// Mitsubishi GX Works2 project: 1 A22-0150 PLC_230728   PLC: Q03UDV

PROGRAM 001  // 現在値ｶｳﾝﾄ
      P100
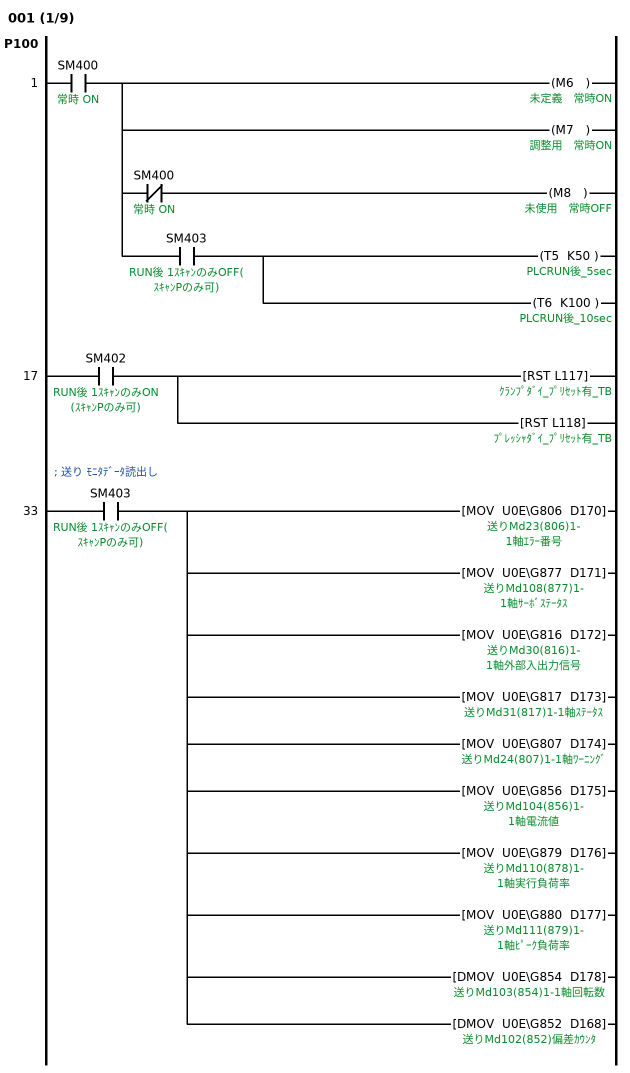
1     LD      SM400  ; 常時 ON
      OUT     M6  ; 未定義　常時ON
      OUT     M7  ; 調整用　常時ON
      MPS
      ANI     SM400  ; 常時 ON
      OUT     M8  ; 未使用　常時OFF
      MPP
      AND     SM403  ; RUN後 1ｽｷｬﾝのみOFF(ｽｷｬﾝPのみ可)
      OUT     T5 K50  ; PLCRUN後_5sec
      OUT     T6 K100  ; PLCRUN後_10sec
17    LD      SM402  ; RUN後 1ｽｷｬﾝのみON (ｽｷｬﾝPのみ可)
      RST     L117  ; ｸﾗﾝﾌﾟﾀﾞｲ_ﾌﾟﾘｾｯﾄ有_TB
      RST     L118  ; ﾌﾟﾚｯｼｬﾀﾞｲ_ﾌﾟﾘｾｯﾄ有_TB
; 
; 送り ﾓﾆﾀﾃﾞｰﾀ読出し
33    LD      SM403  ; RUN後 1ｽｷｬﾝのみOFF(ｽｷｬﾝPのみ可)
      MOV     U0E\G806 D170  ; 送りMd23(806)1-1軸ｴﾗｰ番号
      MOV     U0E\G877 D171  ; 送りMd108(877)1-1軸ｻｰﾎﾞｽﾃｰﾀｽ
      MOV     U0E\G816 D172  ; 送りMd30(816)1-1軸外部入出力信号
      MOV     U0E\G817 D173  ; 送りMd31(817)1-1軸ｽﾃｰﾀｽ
      MOV     U0E\G807 D174  ; 送りMd24(807)1-1軸ﾜｰﾆﾝｸﾞ
      MOV     U0E\G856 D175  ; 送りMd104(856)1-1軸電流値
      MOV     U0E\G879 D176  ; 送りMd110(878)1-1軸実行負荷率
      MOV     U0E\G880 D177  ; 送りMd111(879)1-1軸ﾋﾟｰｸ負荷率
      DMOV    U0E\G854 D178  ; 送りMd103(854)1-1軸回転数
      DMOV    U0E\G852 D168  ; 送りMd102(852)偏差ｶｳﾝﾀ
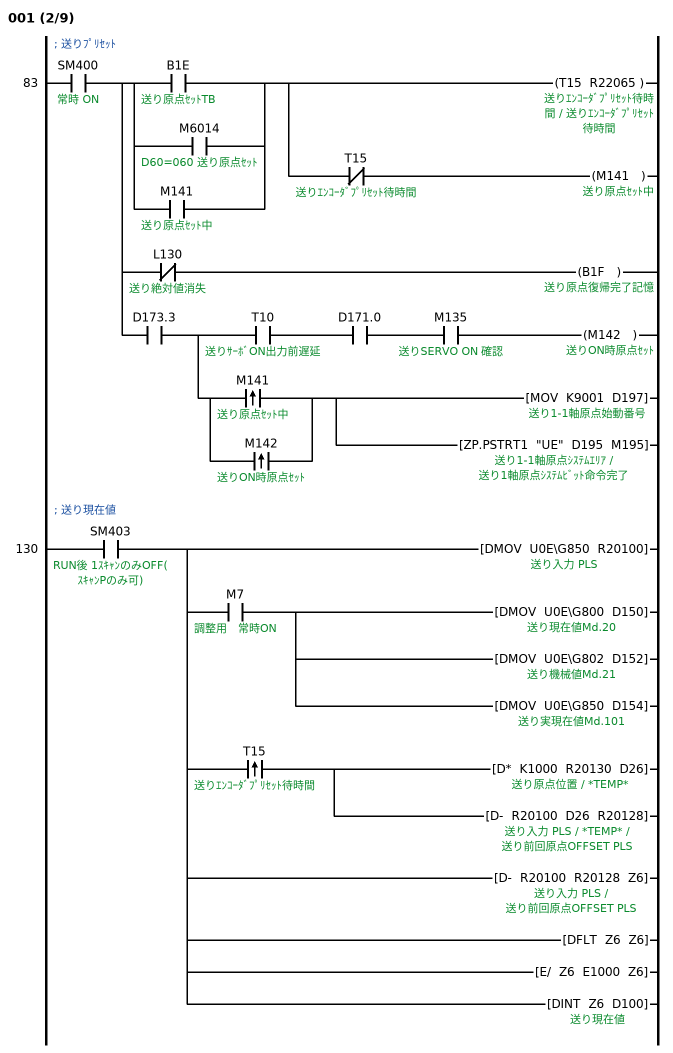
; 
; 送りﾌﾟﾘｾｯﾄ
83    LD      SM400  ; 常時 ON
      MPS
      LD      B1E  ; 送り原点ｾｯﾄTB
      OR      M6014  ; D60=060 送り原点ｾｯﾄ
      OR      M141  ; 送り原点ｾｯﾄ中
      ANB
      OUT     T15 R22065  ; 送りｴﾝｺｰﾀﾞﾌﾟﾘｾｯﾄ待時間 / 送りｴﾝｺｰﾀﾞﾌﾟﾘｾｯﾄ待時間
      ANI     T15  ; 送りｴﾝｺｰﾀﾞﾌﾟﾘｾｯﾄ待時間
      OUT     M141  ; 送り原点ｾｯﾄ中
      MRD
      ANI     L130  ; 送り絶対値消失
      OUT     B1F  ; 送り原点復帰完了記憶
      MPP
      AND     D173.3
      MPS
      AND     T10  ; 送りｻｰﾎﾞON出力前遅延
      AND     D171.0
      AND     M135  ; 送りSERVO ON 確認
      OUT     M142  ; 送りON時原点ｾｯﾄ
      MPP
      LDP     M141  ; 送り原点ｾｯﾄ中
      ORP     M142  ; 送りON時原点ｾｯﾄ
      ANB
      MOV     K9001 D197  ; 送り1-1軸原点始動番号
      ZP.PSTRT1 "UE" D195 M195  ; 送り1-1軸原点ｼｽﾃﾑｴﾘｱ / 送り1軸原点ｼｽﾃﾑﾋﾞｯﾄ命令完了
; 送り現在値
130   LD      SM403  ; RUN後 1ｽｷｬﾝのみOFF(ｽｷｬﾝPのみ可)
      DMOV    U0E\G850 R20100  ; 送り入力 PLS
      MPS
      AND     M7  ; 調整用　常時ON
      DMOV    U0E\G800 D150  ; 送り現在値Md.20
      DMOV    U0E\G802 D152  ; 送り機械値Md.21
      DMOV    U0E\G850 D154  ; 送り実現在値Md.101
      MRD
      ANDP    T15  ; 送りｴﾝｺｰﾀﾞﾌﾟﾘｾｯﾄ待時間
      D*      K1000 R20130 D26  ; 送り原点位置 / *TEMP*
      D-      R20100 D26 R20128  ; 送り前回原点OFFSET PLS
      MPP
      D-      R20100 R20128 Z6
      DFLT    Z6 Z6
      E/      Z6 E1000 Z6
      DINT    Z6 D100  ; 送り現在値
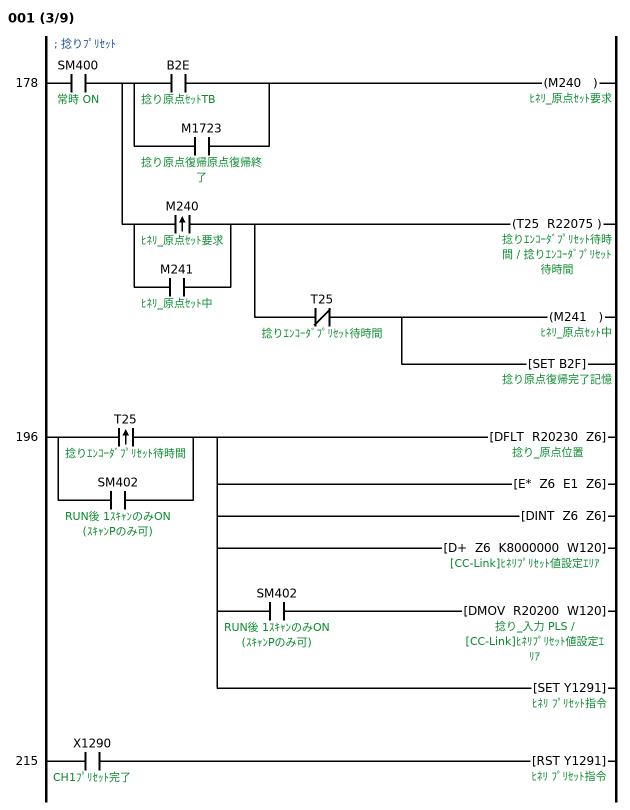
; 
; 捻りﾌﾟﾘｾｯﾄ
178   LD      SM400  ; 常時 ON
      MPS
      LD      B2E  ; 捻り原点ｾｯﾄTB
      OR      M1723  ; 捻り原点復帰原点復帰終了
      ANB
      OUT     M240  ; ﾋﾈﾘ_原点ｾｯﾄ要求
      MPP
      LDP     M240  ; ﾋﾈﾘ_原点ｾｯﾄ要求
      OR      M241  ; ﾋﾈﾘ_原点ｾｯﾄ中
      ANB
      OUT     T25 R22075  ; 捻りｴﾝｺｰﾀﾞﾌﾟﾘｾｯﾄ待時間 / 捻りｴﾝｺｰﾀﾞﾌﾟﾘｾｯﾄ待時間
      ANI     T25  ; 捻りｴﾝｺｰﾀﾞﾌﾟﾘｾｯﾄ待時間
      OUT     M241  ; ﾋﾈﾘ_原点ｾｯﾄ中
      SET     B2F  ; 捻り原点復帰完了記憶
196   LDP     T25  ; 捻りｴﾝｺｰﾀﾞﾌﾟﾘｾｯﾄ待時間
      OR      SM402  ; RUN後 1ｽｷｬﾝのみON (ｽｷｬﾝPのみ可)
      DFLT    R20230 Z6  ; 捻り_原点位置
      E*      Z6 E1 Z6
      DINT    Z6 Z6
      D+      Z6 K8000000 W120  ; [CC-Link]ﾋﾈﾘﾌﾟﾘｾｯﾄ値設定ｴﾘｱ
      MPS
      AND     SM402  ; RUN後 1ｽｷｬﾝのみON (ｽｷｬﾝPのみ可)
      DMOV    R20200 W120  ; 捻り_入力 PLS
      MPP
      SET     Y1291  ; ﾋﾈﾘ ﾌﾟﾘｾｯﾄ指令
215   LD      X1290  ; CH1ﾌﾟﾘｾｯﾄ完了
      RST     Y1291  ; ﾋﾈﾘ ﾌﾟﾘｾｯﾄ指令
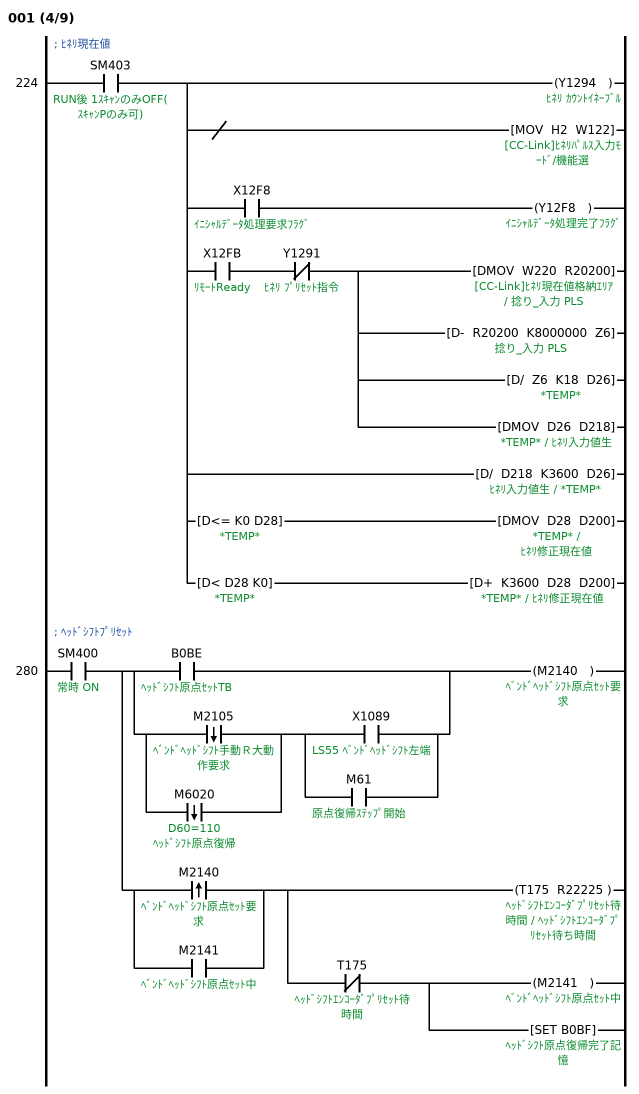
; ﾋﾈﾘ現在値
224   LD      SM403  ; RUN後 1ｽｷｬﾝのみOFF(ｽｷｬﾝPのみ可)
      OUT     Y1294  ; ﾋﾈﾘ ｶｳﾝﾄｲﾈｰﾌﾞﾙ
      MPS
      INV
      MOV     H2 W122  ; [CC-Link]ﾋﾈﾘﾊﾟﾙｽ入力ﾓｰﾄﾞ/機能選
      MRD
      AND     X12F8  ; ｲﾆｼｬﾙﾃﾞｰﾀ処理要求ﾌﾗｸﾞ
      OUT     Y12F8  ; ｲﾆｼｬﾙﾃﾞｰﾀ処理完了ﾌﾗｸﾞ
      MRD
      AND     X12FB  ; ﾘﾓｰﾄReady
      ANI     Y1291  ; ﾋﾈﾘ ﾌﾟﾘｾｯﾄ指令
      DMOV    W220 R20200  ; [CC-Link]ﾋﾈﾘ現在値格納ｴﾘｱ
      D-      R20200 K8000000 Z6
      D/      Z6 K18 D26
      DMOV    D26 D218  ; ﾋﾈﾘ入力値生
      MPP
      D/      D218 K3600 D26
      MPS
      ANDD<=  K0 D28  ; *TEMP*
      DMOV    D28 D200  ; ﾋﾈﾘ修正現在値
      MPP
      ANDD<   D28 K0  ; *TEMP*
      D+      K3600 D28 D200
; 
; ﾍｯﾄﾞｼﾌﾄﾌﾟﾘｾｯﾄ
280   LD      SM400  ; 常時 ON
      MPS
      LD      B0BE  ; ﾍｯﾄﾞｼﾌﾄ原点ｾｯﾄTB
      LDF     M2105  ; ﾍﾞﾝﾄﾞﾍｯﾄﾞｼﾌﾄ手動Ｒ大動作要求
      ORF     M6020  ; D60=110 ﾍｯﾄﾞｼﾌﾄ原点復帰
      LD      X1089  ; LS55 ﾍﾞﾝﾄﾞﾍｯﾄﾞｼﾌﾄ左端
      OR      M61  ; 原点復帰ｽﾃｯﾌﾟ開始
      ANB
      ORB
      ANB
      OUT     M2140  ; ﾍﾞﾝﾄﾞﾍｯﾄﾞｼﾌﾄ原点ｾｯﾄ要求
      MPP
      LDP     M2140  ; ﾍﾞﾝﾄﾞﾍｯﾄﾞｼﾌﾄ原点ｾｯﾄ要求
      OR      M2141  ; ﾍﾞﾝﾄﾞﾍｯﾄﾞｼﾌﾄ原点ｾｯﾄ中
      ANB
      OUT     T175 R22225  ; ﾍｯﾄﾞｼﾌﾄｴﾝｺｰﾀﾞﾌﾟﾘｾｯﾄ待時間 / ﾍｯﾄﾞｼﾌﾄｴﾝｺｰﾀﾞﾌﾟﾘｾｯﾄ待ち時間
      ANI     T175  ; ﾍｯﾄﾞｼﾌﾄｴﾝｺｰﾀﾞﾌﾟﾘｾｯﾄ待時間
      OUT     M2141  ; ﾍﾞﾝﾄﾞﾍｯﾄﾞｼﾌﾄ原点ｾｯﾄ中
      SET     B0BF  ; ﾍｯﾄﾞｼﾌﾄ原点復帰完了記憶
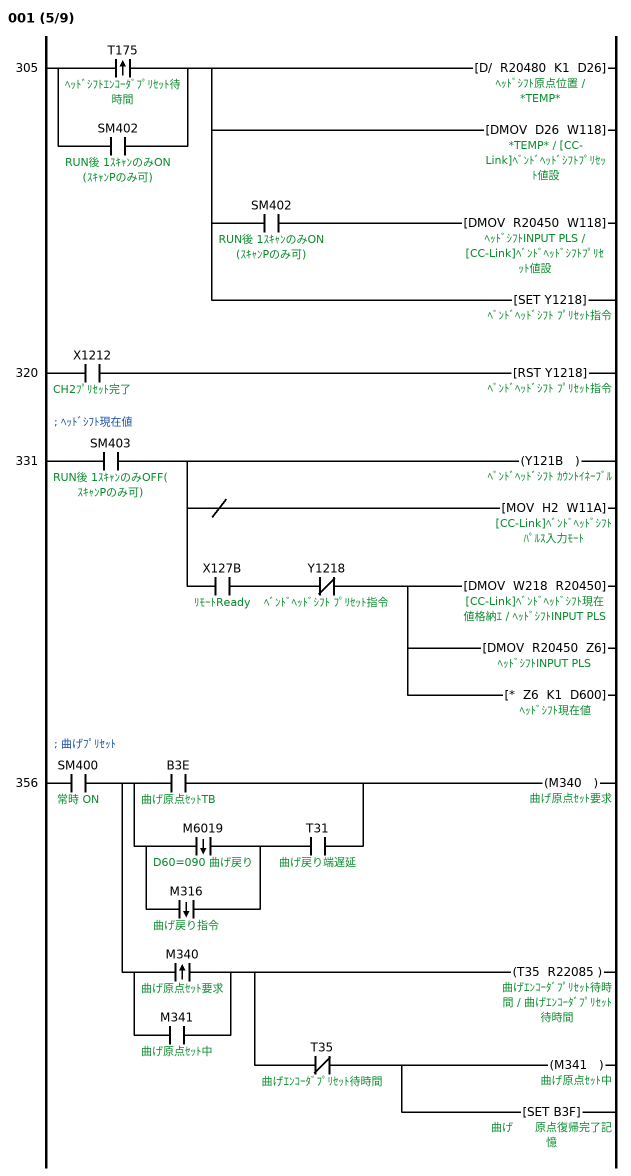
305   LDP     T175  ; ﾍｯﾄﾞｼﾌﾄｴﾝｺｰﾀﾞﾌﾟﾘｾｯﾄ待時間
      OR      SM402  ; RUN後 1ｽｷｬﾝのみON (ｽｷｬﾝPのみ可)
      D/      R20480 K1 D26  ; ﾍｯﾄﾞｼﾌﾄ原点位置
      DMOV    D26 W118  ; [CC-Link]ﾍﾞﾝﾄﾞﾍｯﾄﾞｼﾌﾄﾌﾟﾘｾｯﾄ値設
      MPS
      AND     SM402  ; RUN後 1ｽｷｬﾝのみON (ｽｷｬﾝPのみ可)
      DMOV    R20450 W118  ; ﾍｯﾄﾞｼﾌﾄINPUT PLS
      MPP
      SET     Y1218  ; ﾍﾞﾝﾄﾞﾍｯﾄﾞｼﾌﾄ ﾌﾟﾘｾｯﾄ指令
320   LD      X1212  ; CH2ﾌﾟﾘｾｯﾄ完了
      RST     Y1218  ; ﾍﾞﾝﾄﾞﾍｯﾄﾞｼﾌﾄ ﾌﾟﾘｾｯﾄ指令
; ﾍｯﾄﾞｼﾌﾄ現在値
331   LD      SM403  ; RUN後 1ｽｷｬﾝのみOFF(ｽｷｬﾝPのみ可)
      OUT     Y121B  ; ﾍﾞﾝﾄﾞﾍｯﾄﾞｼﾌﾄ ｶｳﾝﾄｲﾈｰﾌﾞﾙ
      MPS
      INV
      MOV     H2 W11A  ; [CC-Link]ﾍﾞﾝﾄﾞﾍｯﾄﾞｼﾌﾄﾊﾟﾙｽ入力ﾓｰﾄ
      MPP
      AND     X127B  ; ﾘﾓｰﾄReady
      ANI     Y1218  ; ﾍﾞﾝﾄﾞﾍｯﾄﾞｼﾌﾄ ﾌﾟﾘｾｯﾄ指令
      DMOV    W218 R20450  ; [CC-Link]ﾍﾞﾝﾄﾞﾍｯﾄﾞｼﾌﾄ現在値格納ｴ
      DMOV    R20450 Z6
      *       Z6 K1 D600  ; ﾍｯﾄﾞｼﾌﾄ現在値
; 
; 曲げﾌﾟﾘｾｯﾄ
356   LD      SM400  ; 常時 ON
      MPS
      LD      B3E  ; 曲げ原点ｾｯﾄTB
      LDF     M6019  ; D60=090 曲げ戻り
      ORF     M316  ; 曲げ戻り指令
      AND     T31  ; 曲げ戻り端遅延
      ORB
      ANB
      OUT     M340  ; 曲げ原点ｾｯﾄ要求
      MPP
      LDP     M340  ; 曲げ原点ｾｯﾄ要求
      OR      M341  ; 曲げ原点ｾｯﾄ中
      ANB
      OUT     T35 R22085  ; 曲げｴﾝｺｰﾀﾞﾌﾟﾘｾｯﾄ待時間 / 曲げｴﾝｺｰﾀﾞﾌﾟﾘｾｯﾄ待時間
      ANI     T35  ; 曲げｴﾝｺｰﾀﾞﾌﾟﾘｾｯﾄ待時間
      OUT     M341  ; 曲げ原点ｾｯﾄ中
      SET     B3F  ; 曲げ　　原点復帰完了記憶
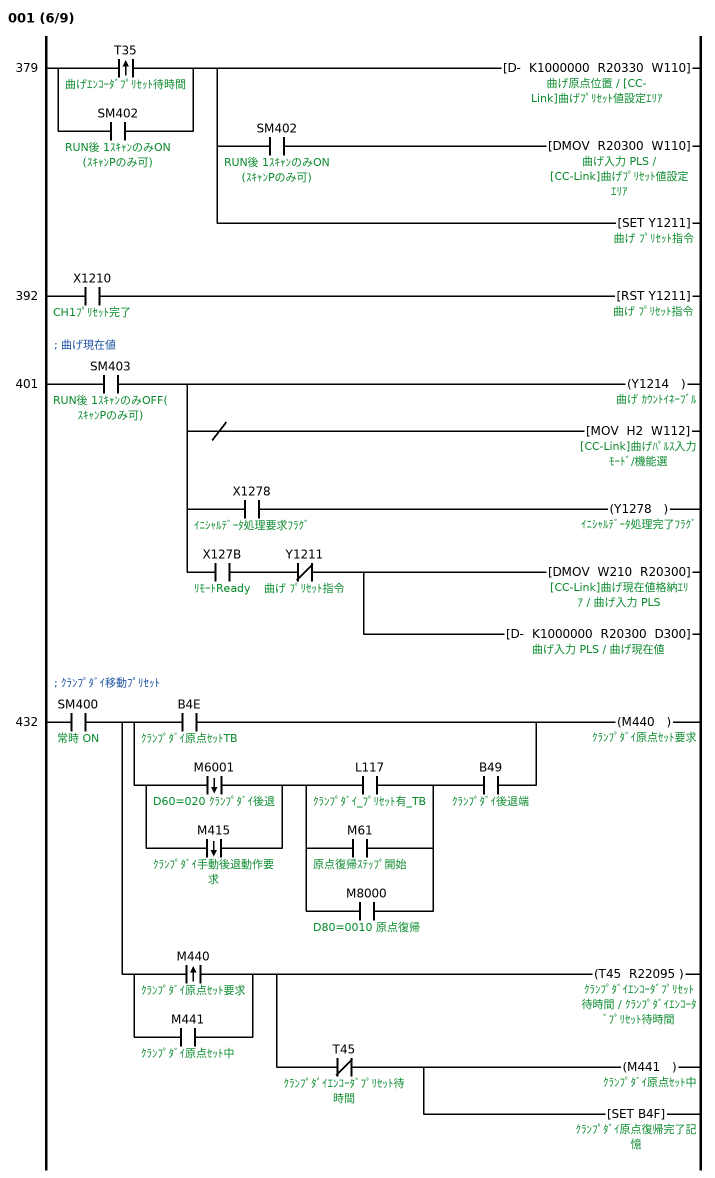
379   LDP     T35  ; 曲げｴﾝｺｰﾀﾞﾌﾟﾘｾｯﾄ待時間
      OR      SM402  ; RUN後 1ｽｷｬﾝのみON (ｽｷｬﾝPのみ可)
      D-      K1000000 R20330 W110  ; 曲げ原点位置 / [CC-Link]曲げﾌﾟﾘｾｯﾄ値設定ｴﾘｱ
      MPS
      AND     SM402  ; RUN後 1ｽｷｬﾝのみON (ｽｷｬﾝPのみ可)
      DMOV    R20300 W110  ; 曲げ入力 PLS
      MPP
      SET     Y1211  ; 曲げ ﾌﾟﾘｾｯﾄ指令
392   LD      X1210  ; CH1ﾌﾟﾘｾｯﾄ完了
      RST     Y1211  ; 曲げ ﾌﾟﾘｾｯﾄ指令
; 曲げ現在値
401   LD      SM403  ; RUN後 1ｽｷｬﾝのみOFF(ｽｷｬﾝPのみ可)
      OUT     Y1214  ; 曲げ ｶｳﾝﾄｲﾈｰﾌﾞﾙ
      MPS
      INV
      MOV     H2 W112  ; [CC-Link]曲げﾊﾟﾙｽ入力ﾓｰﾄﾞ/機能選
      MRD
      AND     X1278  ; ｲﾆｼｬﾙﾃﾞｰﾀ処理要求ﾌﾗｸﾞ
      OUT     Y1278  ; ｲﾆｼｬﾙﾃﾞｰﾀ処理完了ﾌﾗｸﾞ
      MPP
      AND     X127B  ; ﾘﾓｰﾄReady
      ANI     Y1211  ; 曲げ ﾌﾟﾘｾｯﾄ指令
      DMOV    W210 R20300  ; [CC-Link]曲げ現在値格納ｴﾘｱ
      D-      K1000000 R20300 D300  ; 曲げ現在値
; 
; ｸﾗﾝﾌﾟﾀﾞｲ移動ﾌﾟﾘｾｯﾄ
432   LD      SM400  ; 常時 ON
      MPS
      LD      B4E  ; ｸﾗﾝﾌﾟﾀﾞｲ原点ｾｯﾄTB
      LDF     M6001  ; D60=020 ｸﾗﾝﾌﾟﾀﾞｲ後退
      ORF     M415  ; ｸﾗﾝﾌﾟﾀﾞｲ手動後退動作要求
      LD      L117  ; ｸﾗﾝﾌﾟﾀﾞｲ_ﾌﾟﾘｾｯﾄ有_TB
      OR      M61  ; 原点復帰ｽﾃｯﾌﾟ開始
      OR      M8000  ; D80=0010 原点復帰
      ANB
      AND     B49  ; ｸﾗﾝﾌﾟﾀﾞｲ後退端
      ORB
      ANB
      OUT     M440  ; ｸﾗﾝﾌﾟﾀﾞｲ原点ｾｯﾄ要求
      MPP
      LDP     M440  ; ｸﾗﾝﾌﾟﾀﾞｲ原点ｾｯﾄ要求
      OR      M441  ; ｸﾗﾝﾌﾟﾀﾞｲ原点ｾｯﾄ中
      ANB
      OUT     T45 R22095  ; ｸﾗﾝﾌﾟﾀﾞｲｴﾝｺｰﾀﾞﾌﾟﾘｾｯﾄ待時間 / ｸﾗﾝﾌﾟﾀﾞｲｴﾝｺｰﾀﾞﾌﾟﾘｾｯﾄ待時間
      ANI     T45  ; ｸﾗﾝﾌﾟﾀﾞｲｴﾝｺｰﾀﾞﾌﾟﾘｾｯﾄ待時間
      OUT     M441  ; ｸﾗﾝﾌﾟﾀﾞｲ原点ｾｯﾄ中
      SET     B4F  ; ｸﾗﾝﾌﾟﾀﾞｲ原点復帰完了記憶
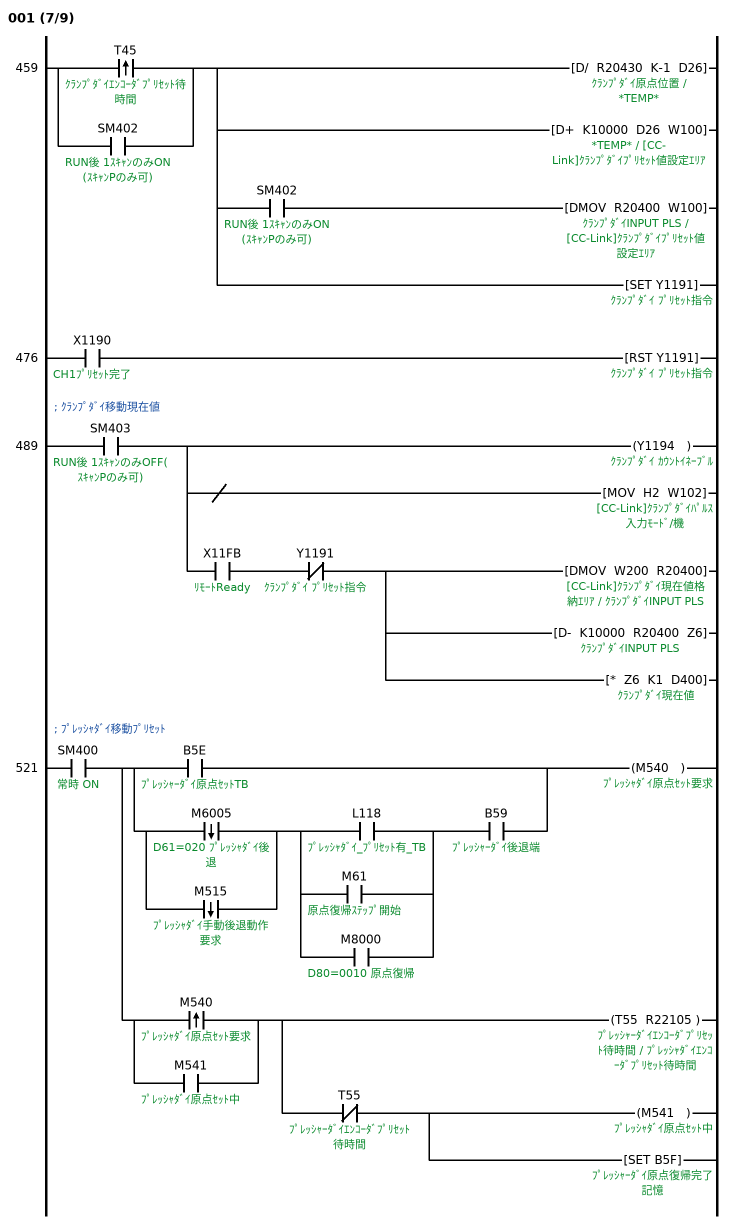
459   LDP     T45  ; ｸﾗﾝﾌﾟﾀﾞｲｴﾝｺｰﾀﾞﾌﾟﾘｾｯﾄ待時間
      OR      SM402  ; RUN後 1ｽｷｬﾝのみON (ｽｷｬﾝPのみ可)
      D/      R20430 K-1 D26  ; ｸﾗﾝﾌﾟﾀﾞｲ原点位置
      D+      K10000 D26 W100  ; [CC-Link]ｸﾗﾝﾌﾟﾀﾞｲﾌﾟﾘｾｯﾄ値設定ｴﾘｱ
      MPS
      AND     SM402  ; RUN後 1ｽｷｬﾝのみON (ｽｷｬﾝPのみ可)
      DMOV    R20400 W100  ; ｸﾗﾝﾌﾟﾀﾞｲINPUT PLS
      MPP
      SET     Y1191  ; ｸﾗﾝﾌﾟﾀﾞｲ ﾌﾟﾘｾｯﾄ指令
476   LD      X1190  ; CH1ﾌﾟﾘｾｯﾄ完了
      RST     Y1191  ; ｸﾗﾝﾌﾟﾀﾞｲ ﾌﾟﾘｾｯﾄ指令
; ｸﾗﾝﾌﾟﾀﾞｲ移動現在値
489   LD      SM403  ; RUN後 1ｽｷｬﾝのみOFF(ｽｷｬﾝPのみ可)
      OUT     Y1194  ; ｸﾗﾝﾌﾟﾀﾞｲ ｶｳﾝﾄｲﾈｰﾌﾞﾙ
      MPS
      INV
      MOV     H2 W102  ; [CC-Link]ｸﾗﾝﾌﾟﾀﾞｲﾊﾟﾙｽ入力ﾓｰﾄﾞ/機
      MPP
      AND     X11FB  ; ﾘﾓｰﾄReady
      ANI     Y1191  ; ｸﾗﾝﾌﾟﾀﾞｲ ﾌﾟﾘｾｯﾄ指令
      DMOV    W200 R20400  ; [CC-Link]ｸﾗﾝﾌﾟﾀﾞｲ現在値格納ｴﾘｱ
      D-      K10000 R20400 Z6
      *       Z6 K1 D400  ; ｸﾗﾝﾌﾟﾀﾞｲ現在値
; 
; ﾌﾟﾚｯｼｬﾀﾞｲ移動ﾌﾟﾘｾｯﾄ
521   LD      SM400  ; 常時 ON
      MPS
      LD      B5E  ; ﾌﾟﾚｯｼｬｰﾀﾞｲ原点ｾｯﾄTB
      LDF     M6005  ; D61=020 ﾌﾟﾚｯｼｬﾀﾞｲ後退
      ORF     M515  ; ﾌﾟﾚｯｼｬﾀﾞｲ手動後退動作要求
      LD      L118  ; ﾌﾟﾚｯｼｬﾀﾞｲ_ﾌﾟﾘｾｯﾄ有_TB
      OR      M61  ; 原点復帰ｽﾃｯﾌﾟ開始
      OR      M8000  ; D80=0010 原点復帰
      ANB
      AND     B59  ; ﾌﾟﾚｯｼｬｰﾀﾞｲ後退端
      ORB
      ANB
      OUT     M540  ; ﾌﾟﾚｯｼｬﾀﾞｲ原点ｾｯﾄ要求
      MPP
      LDP     M540  ; ﾌﾟﾚｯｼｬﾀﾞｲ原点ｾｯﾄ要求
      OR      M541  ; ﾌﾟﾚｯｼｬﾀﾞｲ原点ｾｯﾄ中
      ANB
      OUT     T55 R22105  ; ﾌﾟﾚｯｼｬｰﾀﾞｲｴﾝｺｰﾀﾞﾌﾟﾘｾｯﾄ待時間 / ﾌﾟﾚｯｼｬﾀﾞｲｴﾝｺｰﾀﾞﾌﾟﾘｾｯﾄ待時間
      ANI     T55  ; ﾌﾟﾚｯｼｬｰﾀﾞｲｴﾝｺｰﾀﾞﾌﾟﾘｾｯﾄ待時間
      OUT     M541  ; ﾌﾟﾚｯｼｬﾀﾞｲ原点ｾｯﾄ中
      SET     B5F  ; ﾌﾟﾚｯｼｬｰﾀﾞｲ原点復帰完了記憶
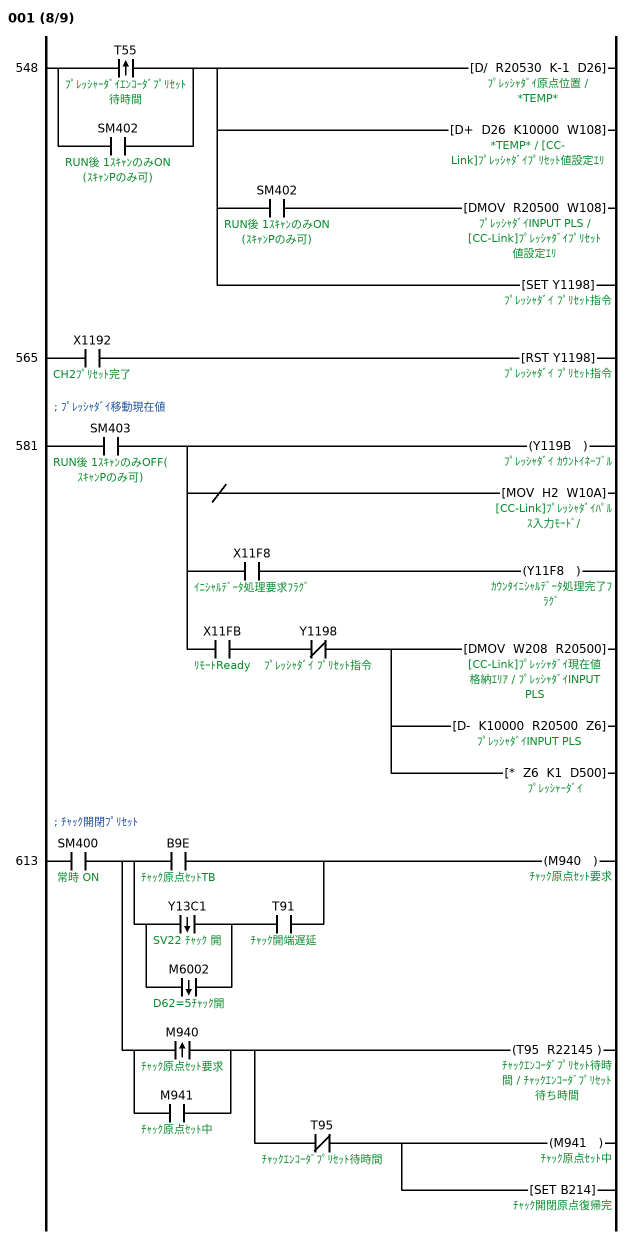
548   LDP     T55  ; ﾌﾟﾚｯｼｬｰﾀﾞｲｴﾝｺｰﾀﾞﾌﾟﾘｾｯﾄ待時間
      OR      SM402  ; RUN後 1ｽｷｬﾝのみON (ｽｷｬﾝPのみ可)
      D/      R20530 K-1 D26  ; ﾌﾟﾚｯｼｬﾀﾞｲ原点位置
      D+      D26 K10000 W108  ; [CC-Link]ﾌﾟﾚｯｼｬﾀﾞｲﾌﾟﾘｾｯﾄ値設定ｴﾘ
      MPS
      AND     SM402  ; RUN後 1ｽｷｬﾝのみON (ｽｷｬﾝPのみ可)
      DMOV    R20500 W108  ; ﾌﾟﾚｯｼｬﾀﾞｲINPUT PLS
      MPP
      SET     Y1198  ; ﾌﾟﾚｯｼｬﾀﾞｲ ﾌﾟﾘｾｯﾄ指令
565   LD      X1192  ; CH2ﾌﾟﾘｾｯﾄ完了
      RST     Y1198  ; ﾌﾟﾚｯｼｬﾀﾞｲ ﾌﾟﾘｾｯﾄ指令
; 
; ﾌﾟﾚｯｼｬﾀﾞｲ移動現在値
581   LD      SM403  ; RUN後 1ｽｷｬﾝのみOFF(ｽｷｬﾝPのみ可)
      OUT     Y119B  ; ﾌﾟﾚｯｼｬﾀﾞｲ ｶｳﾝﾄｲﾈｰﾌﾞﾙ
      MPS
      INV
      MOV     H2 W10A  ; [CC-Link]ﾌﾟﾚｯｼｬﾀﾞｲﾊﾟﾙｽ入力ﾓｰﾄﾞ/
      MRD
      AND     X11F8  ; ｲﾆｼｬﾙﾃﾞｰﾀ処理要求ﾌﾗｸﾞ
      OUT     Y11F8  ; ｶｳﾝﾀｲﾆｼｬﾙﾃﾞｰﾀ処理完了ﾌﾗｸﾞ
      MPP
      AND     X11FB  ; ﾘﾓｰﾄReady
      ANI     Y1198  ; ﾌﾟﾚｯｼｬﾀﾞｲ ﾌﾟﾘｾｯﾄ指令
      DMOV    W208 R20500  ; [CC-Link]ﾌﾟﾚｯｼｬﾀﾞｲ現在値格納ｴﾘｱ
      D-      K10000 R20500 Z6
      *       Z6 K1 D500  ; ﾌﾟﾚｯｼｬｰﾀﾞｲ
; 
; ﾁｬｯｸ開閉ﾌﾟﾘｾｯﾄ
613   LD      SM400  ; 常時 ON
      MPS
      LD      B9E  ; ﾁｬｯｸ原点ｾｯﾄTB
      LDF     Y13C1  ; SV22 ﾁｬｯｸ 開
      ORF     M6002  ; D62=5ﾁｬｯｸ開
      AND     T91  ; ﾁｬｯｸ開端遅延
      ORB
      ANB
      OUT     M940  ; ﾁｬｯｸ原点ｾｯﾄ要求
      MPP
      LDP     M940  ; ﾁｬｯｸ原点ｾｯﾄ要求
      OR      M941  ; ﾁｬｯｸ原点ｾｯﾄ中
      ANB
      OUT     T95 R22145  ; ﾁｬｯｸｴﾝｺｰﾀﾞﾌﾟﾘｾｯﾄ待時間 / ﾁｬｯｸｴﾝｺｰﾀﾞﾌﾟﾘｾｯﾄ待ち時間
      ANI     T95  ; ﾁｬｯｸｴﾝｺｰﾀﾞﾌﾟﾘｾｯﾄ待時間
      OUT     M941  ; ﾁｬｯｸ原点ｾｯﾄ中
      SET     B214  ; ﾁｬｯｸ開閉原点復帰完
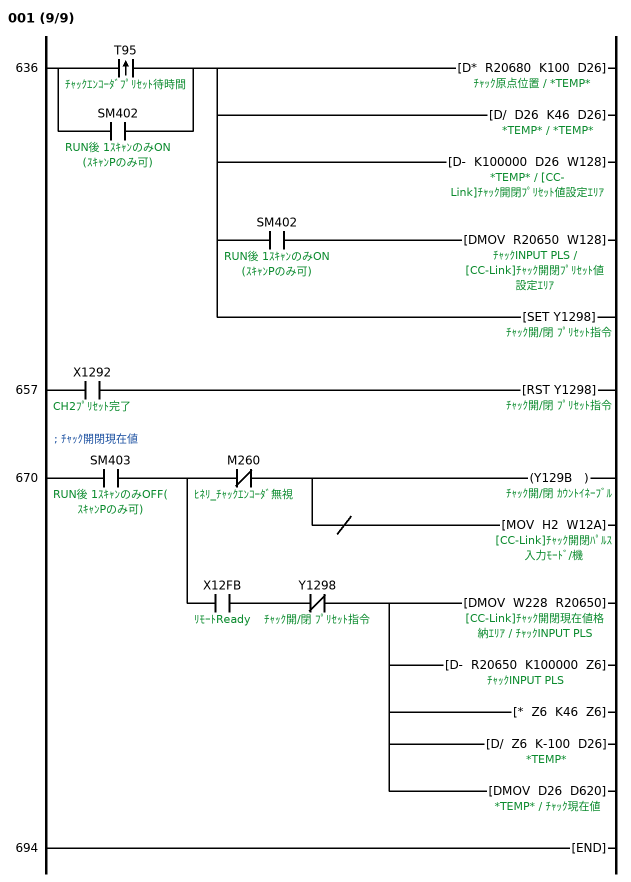
636   LDP     T95  ; ﾁｬｯｸｴﾝｺｰﾀﾞﾌﾟﾘｾｯﾄ待時間
      OR      SM402  ; RUN後 1ｽｷｬﾝのみON (ｽｷｬﾝPのみ可)
      D*      R20680 K100 D26  ; ﾁｬｯｸ原点位置
      D/      D26 K46 D26
      D-      K100000 D26 W128  ; [CC-Link]ﾁｬｯｸ開閉ﾌﾟﾘｾｯﾄ値設定ｴﾘｱ
      MPS
      AND     SM402  ; RUN後 1ｽｷｬﾝのみON (ｽｷｬﾝPのみ可)
      DMOV    R20650 W128  ; ﾁｬｯｸINPUT PLS
      MPP
      SET     Y1298  ; ﾁｬｯｸ開/閉 ﾌﾟﾘｾｯﾄ指令
657   LD      X1292  ; CH2ﾌﾟﾘｾｯﾄ完了
      RST     Y1298  ; ﾁｬｯｸ開/閉 ﾌﾟﾘｾｯﾄ指令
; 
; ﾁｬｯｸ開閉現在値
670   LD      SM403  ; RUN後 1ｽｷｬﾝのみOFF(ｽｷｬﾝPのみ可)
      MPS
      ANI     M260  ; ﾋﾈﾘ_ﾁｬｯｸｴﾝｺｰﾀﾞ無視
      OUT     Y129B  ; ﾁｬｯｸ開/閉 ｶｳﾝﾄｲﾈｰﾌﾞﾙ
      INV
      MOV     H2 W12A  ; [CC-Link]ﾁｬｯｸ開閉ﾊﾟﾙｽ入力ﾓｰﾄﾞ/機
      MPP
      AND     X12FB  ; ﾘﾓｰﾄReady
      ANI     Y1298  ; ﾁｬｯｸ開/閉 ﾌﾟﾘｾｯﾄ指令
      DMOV    W228 R20650  ; [CC-Link]ﾁｬｯｸ開閉現在値格納ｴﾘｱ
      D-      R20650 K100000 Z6
      *       Z6 K46 Z6
      D/      Z6 K-100 D26
      DMOV    D26 D620  ; ﾁｬｯｸ現在値
694   END
END_PROGRAM

PROGRAM 002  // 状態検出
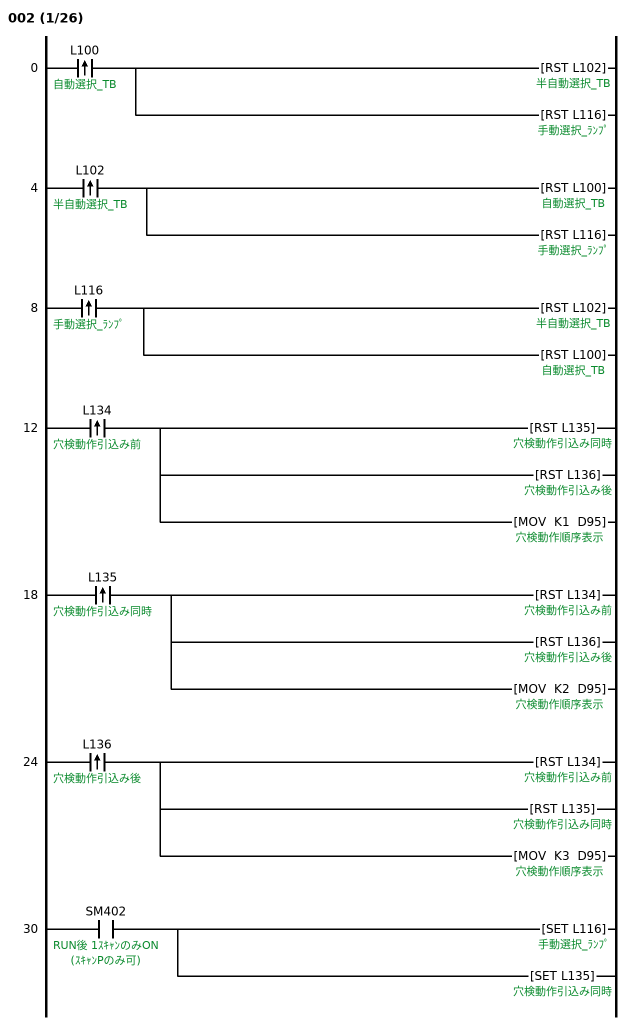
0     LDP     L100  ; 自動選択_TB
      RST     L102  ; 半自動選択_TB
      RST     L116  ; 手動選択_ﾗﾝﾌﾟ
4     LDP     L102  ; 半自動選択_TB
      RST     L100  ; 自動選択_TB
      RST     L116  ; 手動選択_ﾗﾝﾌﾟ
8     LDP     L116  ; 手動選択_ﾗﾝﾌﾟ
      RST     L102  ; 半自動選択_TB
      RST     L100  ; 自動選択_TB
12    LDP     L134  ; 穴検動作引込み前
      RST     L135  ; 穴検動作引込み同時
      RST     L136  ; 穴検動作引込み後
      MOV     K1 D95  ; 穴検動作順序表示
18    LDP     L135  ; 穴検動作引込み同時
      RST     L134  ; 穴検動作引込み前
      RST     L136  ; 穴検動作引込み後
      MOV     K2 D95
24    LDP     L136  ; 穴検動作引込み後
      RST     L134  ; 穴検動作引込み前
      RST     L135  ; 穴検動作引込み同時
      MOV     K3 D95
30    LD      SM402  ; RUN後 1ｽｷｬﾝのみON (ｽｷｬﾝPのみ可)
      SET     L116  ; 手動選択_ﾗﾝﾌﾟ
      SET     L135  ; 穴検動作引込み同時
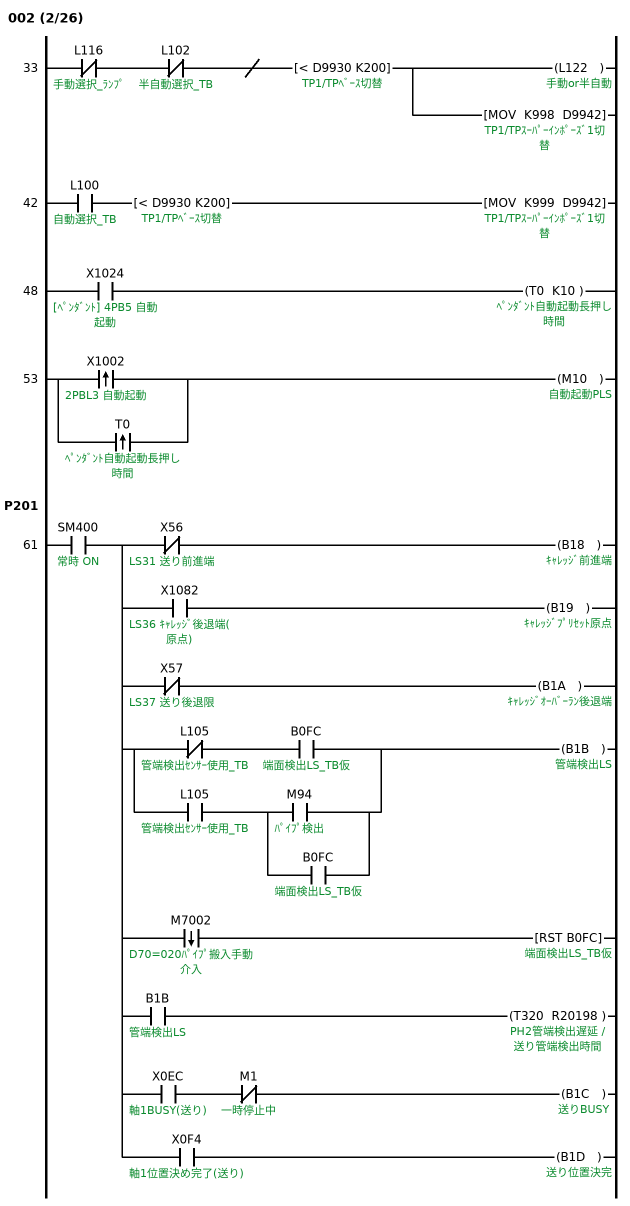
33    LDI     L116  ; 手動選択_ﾗﾝﾌﾟ
      ANI     L102  ; 半自動選択_TB
      INV
      AND<    D9930 K200  ; TP1/TPﾍﾞｰｽ切替
      OUT     L122  ; 手動or半自動
      MOV     K998 D9942  ; TP1/TPｽｰﾊﾟｰｲﾝﾎﾟｰｽﾞ1切替
42    LD      L100  ; 自動選択_TB
      AND<    D9930 K200  ; TP1/TPﾍﾞｰｽ切替
      MOV     K999 D9942
48    LD      X1024  ; [ﾍﾟﾝﾀﾞﾝﾄ] 4PB5 自動 起動
      OUT     T0 K10  ; ﾍﾟﾝﾀﾞﾝﾄ自動起動長押し時間
53    LDP     X1002  ; 2PBL3 自動起動
      ORP     T0  ; ﾍﾟﾝﾀﾞﾝﾄ自動起動長押し時間
      OUT     M10  ; 自動起動PLS
; 
      P201
61    LD      SM400  ; 常時 ON
      MPS
      ANI     X56  ; LS31 送り前進端
      OUT     B18  ; ｷｬﾚｯｼﾞ前進端
      MRD
      AND     X1082  ; LS36 ｷｬﾚｯｼﾞ後退端(原点)
      OUT     B19  ; ｷｬﾚｯｼﾞﾌﾟﾘｾｯﾄ原点
      MRD
      ANI     X57  ; LS37 送り後退限
      OUT     B1A  ; ｷｬﾚｯｼﾞｵｰﾊﾞｰﾗﾝ後退端
      MRD
      LDI     L105  ; 管端検出ｾﾝｻｰ使用_TB
      AND     B0FC  ; 端面検出LS_TB仮
      LD      L105  ; 管端検出ｾﾝｻｰ使用_TB
      LD      M94  ; ﾊﾟｲﾌﾟ検出
      OR      B0FC  ; 端面検出LS_TB仮
      ANB
      ORB
      ANB
      OUT     B1B  ; 管端検出LS
      MRD
      ANDF    M7002  ; D70=020ﾊﾟｲﾌﾟ搬入手動介入
      RST     B0FC  ; 端面検出LS_TB仮
      MRD
      AND     B1B  ; 管端検出LS
      OUT     T320 R20198  ; PH2管端検出遅延 / 送り管端検出時間
      MRD
      AND     X0EC  ; 軸1BUSY(送り)
      ANI     M1  ; 一時停止中
      OUT     B1C  ; 送りBUSY
      MPP
      AND     X0F4  ; 軸1位置決め完了(送り)
      OUT     B1D  ; 送り位置決完
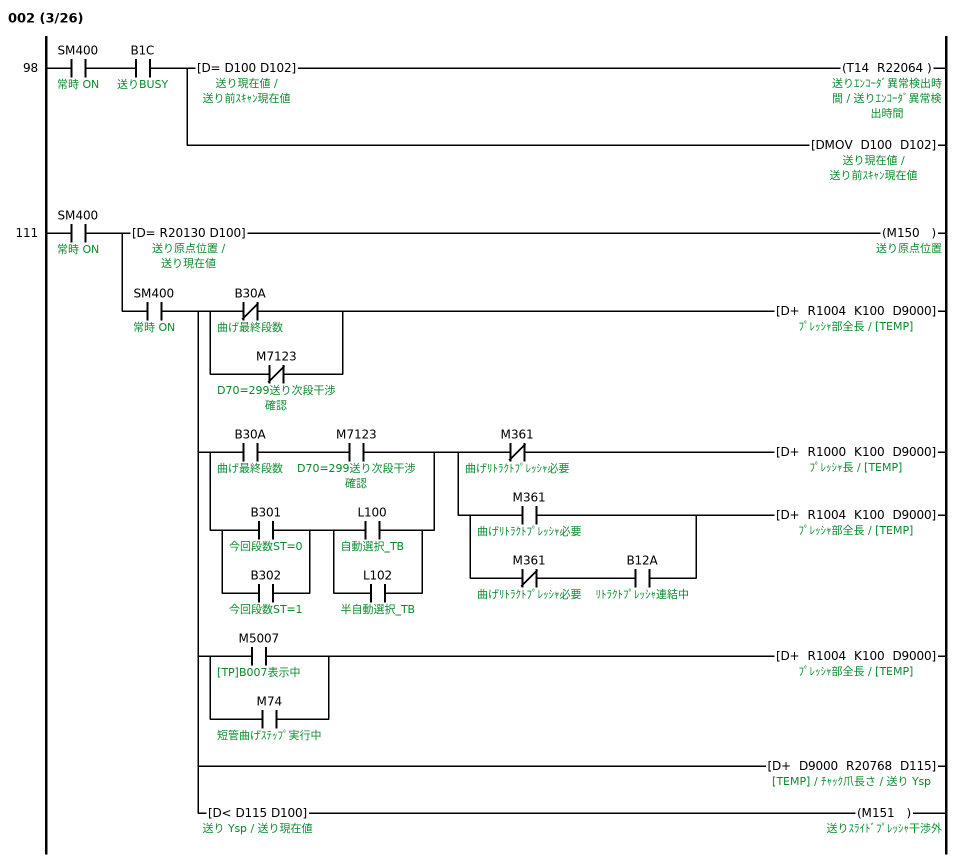
98    LD      SM400  ; 常時 ON
      AND     B1C  ; 送りBUSY
      MPS
      ANDD=   D100 D102  ; 送り現在値 / 送り前ｽｷｬﾝ現在値
      OUT     T14 R22064  ; 送りｴﾝｺｰﾀﾞ異常検出時間 / 送りｴﾝｺｰﾀﾞ異常検出時間
      MPP
      DMOV    D100 D102
111   LD      SM400  ; 常時 ON
      MPS
      ANDD=   R20130 D100  ; 送り原点位置 / 送り現在値
      OUT     M150  ; 送り原点位置
      MPP
      AND     SM400  ; 常時 ON
      MPS
      LDI     B30A  ; 曲げ最終段数
      ORI     M7123  ; D70=299送り次段干渉確認
      ANB
      D+      R1004 K100 D9000  ; ﾌﾟﾚｯｼｬ部全長 / [TEMP]
      MRD
      LD      B30A  ; 曲げ最終段数
      AND     M7123  ; D70=299送り次段干渉確認
      LD      B301  ; 今回段数ST=0
      OR      B302  ; 今回段数ST=1
      LD      L100  ; 自動選択_TB
      OR      L102  ; 半自動選択_TB
      ANB
      ORB
      ANB
      MPS
      ANI     M361  ; 曲げﾘﾄﾗｸﾄﾌﾟﾚｯｼｬ必要
      D+      R1000 K100 D9000  ; ﾌﾟﾚｯｼｬ長
      MPP
      LD      M361  ; 曲げﾘﾄﾗｸﾄﾌﾟﾚｯｼｬ必要
      LDI     M361  ; 曲げﾘﾄﾗｸﾄﾌﾟﾚｯｼｬ必要
      AND     B12A  ; ﾘﾄﾗｸﾄﾌﾟﾚｯｼｬ連結中
      ORB
      ANB
      D+      R1004 K100 D9000
      MRD
      LD      M5007  ; [TP]B007表示中
      OR      M74  ; 短管曲げｽﾃｯﾌﾟ実行中
      ANB
      D+      R1004 K100 D9000
      MPP
      D+      D9000 R20768 D115  ; ﾁｬｯｸ爪長さ / 送り Ysp
      ANDD<   D115 D100  ; 送り Ysp / 送り現在値
      OUT     M151  ; 送りｽﾗｲﾄﾞﾌﾟﾚｯｼｬ干渉外
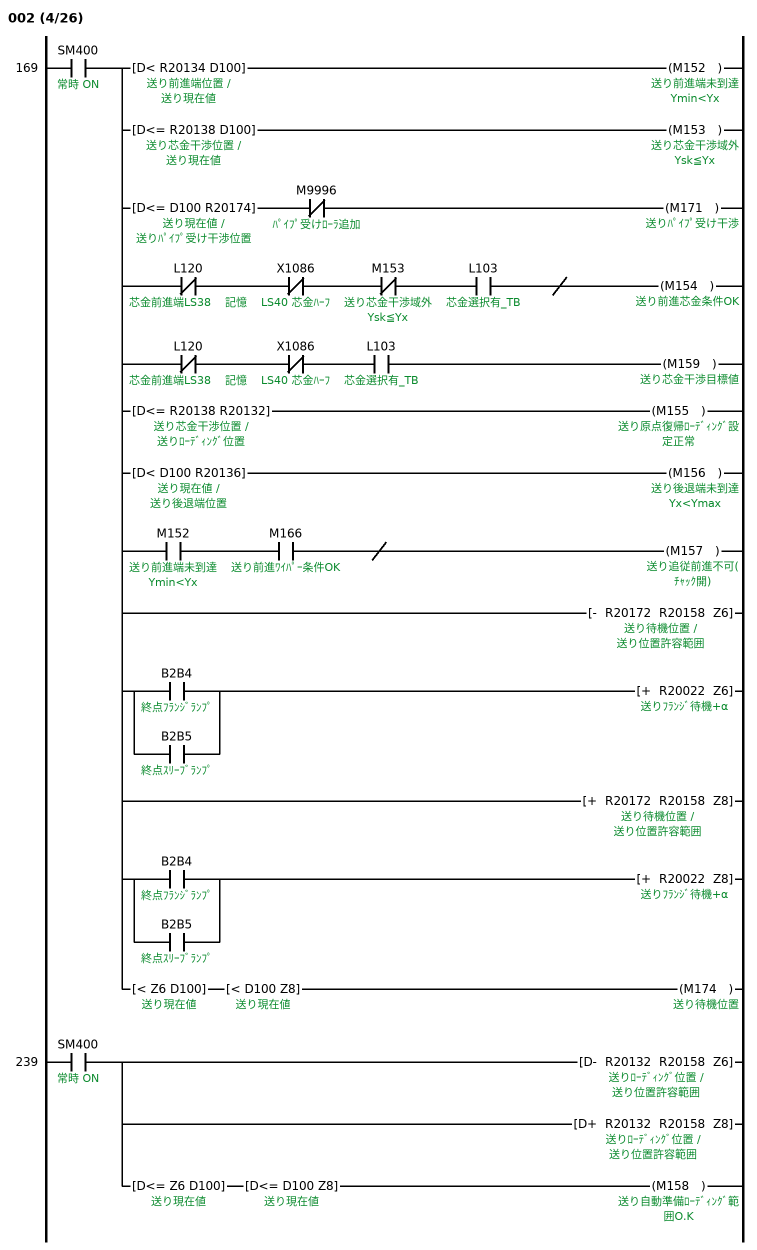
169   LD      SM400  ; 常時 ON
      MPS
      ANDD<   R20134 D100  ; 送り前進端位置 / 送り現在値
      OUT     M152  ; 送り前進端未到達 Ymin<Yx
      MRD
      ANDD<=  R20138 D100  ; 送り芯金干渉位置 / 送り現在値
      OUT     M153  ; 送り芯金干渉域外 Ysk≦Yx
      MRD
      ANDD<=  D100 R20174  ; 送り現在値 / 送りﾊﾟｲﾌﾟ受け干渉位置
      ANI     M9996  ; ﾊﾟｲﾌﾟ受けﾛｰﾗ追加
      OUT     M171  ; 送りﾊﾟｲﾌﾟ受け干渉
      MRD
      ANI     L120  ; 芯金前進端LS38    記憶
      ANI     X1086  ; LS40 芯金ﾊｰﾌ
      ANI     M153  ; 送り芯金干渉域外 Ysk≦Yx
      AND     L103  ; 芯金選択有_TB
      INV
      OUT     M154  ; 送り前進芯金条件OK
      MRD
      ANI     L120  ; 芯金前進端LS38    記憶
      ANI     X1086  ; LS40 芯金ﾊｰﾌ
      AND     L103  ; 芯金選択有_TB
      OUT     M159  ; 送り芯金干渉目標値
      MRD
      ANDD<=  R20138 R20132  ; 送り芯金干渉位置 / 送りﾛｰﾃﾞｨﾝｸﾞ位置
      OUT     M155  ; 送り原点復帰ﾛｰﾃﾞｨﾝｸﾞ設定正常
      MRD
      ANDD<   D100 R20136  ; 送り現在値 / 送り後退端位置
      OUT     M156  ; 送り後退端未到達 Yx<Ymax
      MRD
      AND     M152  ; 送り前進端未到達 Ymin<Yx
      AND     M166  ; 送り前進ﾜｲﾊﾟｰ条件OK
      INV
      OUT     M157  ; 送り追従前進不可(ﾁｬｯｸ開)
      MPP
      -       R20172 R20158 Z6  ; 送り待機位置 / 送り位置許容範囲
      MPS
      LD      B2B4  ; 終点ﾌﾗﾝｼﾞﾗﾝﾌﾟ
      OR      B2B5  ; 終点ｽﾘｰﾌﾞﾗﾝﾌﾟ
      ANB
      +       R20022 Z6  ; 送りﾌﾗﾝｼﾞ待機+α
      MPP
      +       R20172 R20158 Z8
      MPS
      LD      B2B4  ; 終点ﾌﾗﾝｼﾞﾗﾝﾌﾟ
      OR      B2B5  ; 終点ｽﾘｰﾌﾞﾗﾝﾌﾟ
      ANB
      +       R20022 Z8
      MPP
      AND<    Z6 D100  ; 送り現在値
      AND<    D100 Z8  ; 送り現在値
      OUT     M174  ; 送り待機位置
239   LD      SM400  ; 常時 ON
      D-      R20132 R20158 Z6
      D+      R20132 R20158 Z8
      ANDD<=  Z6 D100  ; 送り現在値
      ANDD<=  D100 Z8  ; 送り現在値
      OUT     M158  ; 送り自動準備ﾛｰﾃﾞｨﾝｸﾞ範囲O.K
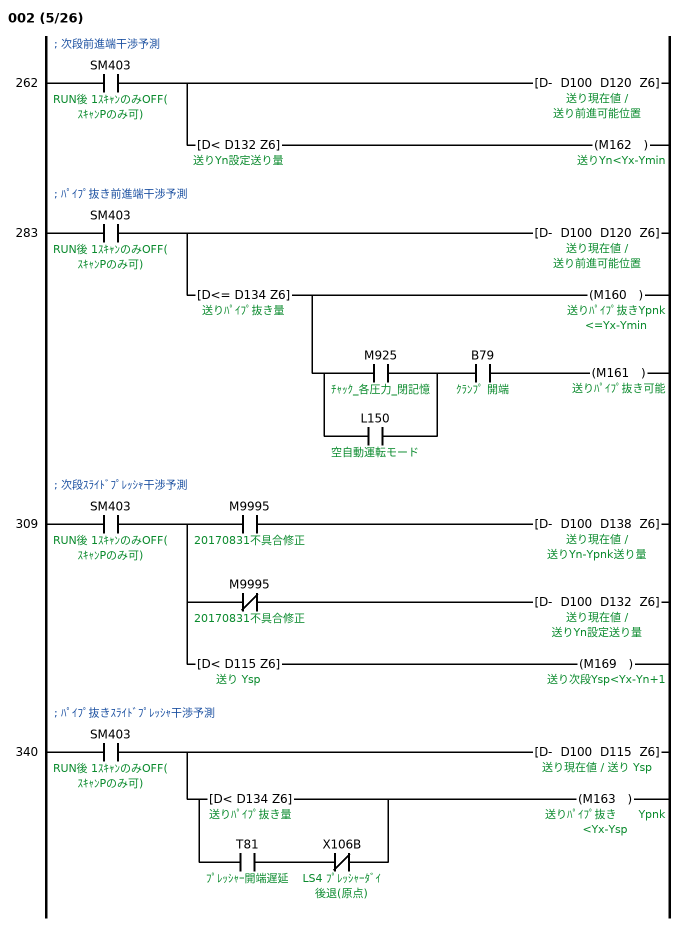
; 次段前進端干渉予測
262   LD      SM403  ; RUN後 1ｽｷｬﾝのみOFF(ｽｷｬﾝPのみ可)
      D-      D100 D120 Z6  ; 送り前進可能位置
      ANDD<   D132 Z6  ; 送りYn設定送り量
      OUT     M162  ; 送りYn<Yx-Ymin
; ﾊﾟｲﾌﾟ抜き前進端干渉予測
283   LD      SM403  ; RUN後 1ｽｷｬﾝのみOFF(ｽｷｬﾝPのみ可)
      D-      D100 D120 Z6
      ANDD<=  D134 Z6  ; 送りﾊﾟｲﾌﾟ抜き量
      OUT     M160  ; 送りﾊﾟｲﾌﾟ抜きYpnk <=Yx-Ymin
      LD      M925  ; ﾁｬｯｸ_各圧力_閉記憶
      OR      L150  ; 空自動運転モード
      ANB
      AND     B79  ; ｸﾗﾝﾌﾟ 開端
      OUT     M161  ; 送りﾊﾟｲﾌﾟ抜き可能
; 次段ｽﾗｲﾄﾞﾌﾟﾚｯｼｬ干渉予測
309   LD      SM403  ; RUN後 1ｽｷｬﾝのみOFF(ｽｷｬﾝPのみ可)
      MPS
      AND     M9995  ; 20170831不具合修正
      D-      D100 D138 Z6  ; 送りYn-Ypnk送り量
      MRD
      ANI     M9995  ; 20170831不具合修正
      D-      D100 D132 Z6
      MPP
      ANDD<   D115 Z6  ; 送り Ysp
      OUT     M169  ; 送り次段Ysp<Yx-Yn+1
; ﾊﾟｲﾌﾟ抜きｽﾗｲﾄﾞﾌﾟﾚｯｼｬ干渉予測
340   LD      SM403  ; RUN後 1ｽｷｬﾝのみOFF(ｽｷｬﾝPのみ可)
      D-      D100 D115 Z6
      LDD<    D134 Z6  ; 送りﾊﾟｲﾌﾟ抜き量
      LD      T81  ; ﾌﾟﾚｯｼｬｰ開端遅延
      ANI     X106B  ; LS4 ﾌﾟﾚｯｼｬｰﾀﾞｲ 後退(原点)
      ORB
      ANB
      OUT     M163  ; 送りﾊﾟｲﾌﾟ抜き　　Ypnk<Yx-Ysp
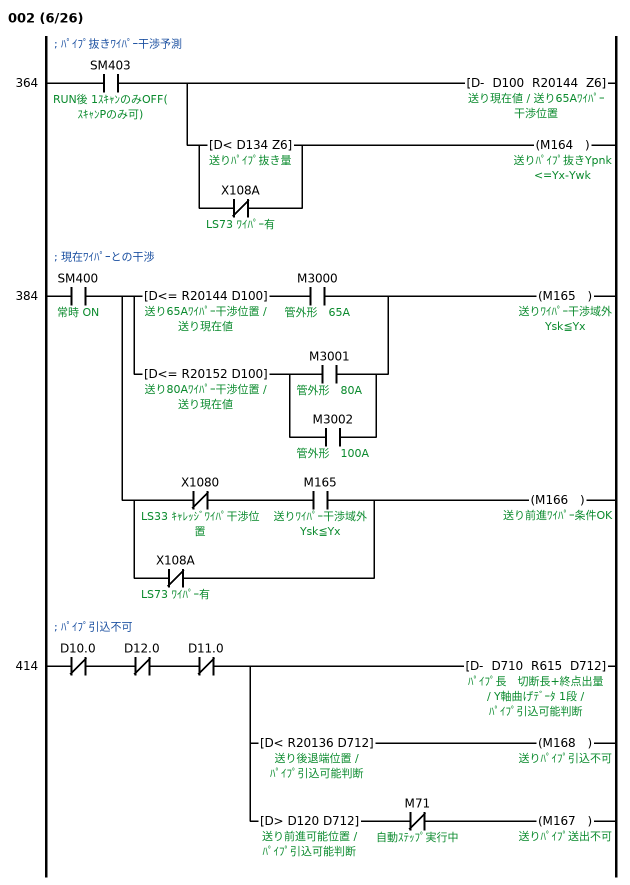
; ﾊﾟｲﾌﾟ抜きﾜｲﾊﾟｰ干渉予測
364   LD      SM403  ; RUN後 1ｽｷｬﾝのみOFF(ｽｷｬﾝPのみ可)
      D-      D100 R20144 Z6  ; 送り65Aﾜｲﾊﾟｰ干渉位置
      LDD<    D134 Z6  ; 送りﾊﾟｲﾌﾟ抜き量
      ORI     X108A  ; LS73 ﾜｲﾊﾟｰ有
      ANB
      OUT     M164  ; 送りﾊﾟｲﾌﾟ抜きYpnk <=Yx-Ywk
; 現在ﾜｲﾊﾟｰとの干渉
384   LD      SM400  ; 常時 ON
      MPS
      LDD<=   R20144 D100  ; 送り65Aﾜｲﾊﾟｰ干渉位置 / 送り現在値
      AND     M3000  ; 管外形　65A
      LDD<=   R20152 D100  ; 送り80Aﾜｲﾊﾟｰ干渉位置 / 送り現在値
      LD      M3001  ; 管外形　80A
      OR      M3002  ; 管外形　100A
      ANB
      ORB
      ANB
      OUT     M165  ; 送りﾜｲﾊﾟｰ干渉域外 Ysk≦Yx
      MPP
      LDI     X1080  ; LS33 ｷｬﾚｯｼﾞﾜｲﾊﾟ干渉位置
      AND     M165  ; 送りﾜｲﾊﾟｰ干渉域外 Ysk≦Yx
      ORI     X108A  ; LS73 ﾜｲﾊﾟｰ有
      ANB
      OUT     M166  ; 送り前進ﾜｲﾊﾟｰ条件OK
; ﾊﾟｲﾌﾟ引込不可
414   LDI     D10.0
      ANI     D12.0
      ANI     D11.0
      D-      D710 R615 D712  ; ﾊﾟｲﾌﾟ長　切断長+終点出量 / Y軸曲げﾃﾞｰﾀ 1段 / ﾊﾟｲﾌﾟ引込可能判断
      MPS
      ANDD<   R20136 D712  ; 送り後退端位置 / ﾊﾟｲﾌﾟ引込可能判断
      OUT     M168  ; 送りﾊﾟｲﾌﾟ引込不可
      MPP
      ANDD>   D120 D712  ; 送り前進可能位置 / ﾊﾟｲﾌﾟ引込可能判断
      ANI     M71  ; 自動ｽﾃｯﾌﾟ実行中
      OUT     M167  ; 送りﾊﾟｲﾌﾟ送出不可
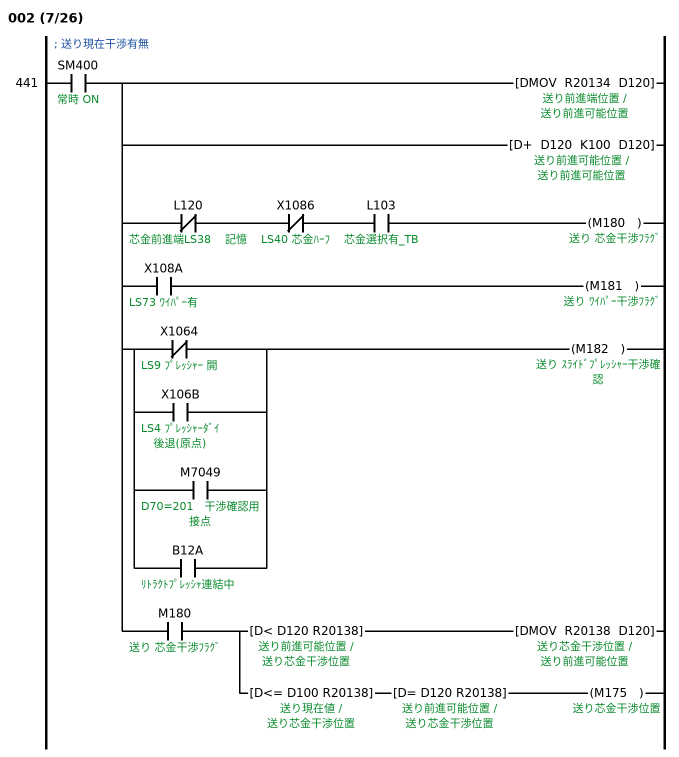
; 送り現在干渉有無
441   LD      SM400  ; 常時 ON
      DMOV    R20134 D120
      D+      D120 K100 D120
      MPS
      ANI     L120  ; 芯金前進端LS38    記憶
      ANI     X1086  ; LS40 芯金ﾊｰﾌ
      AND     L103  ; 芯金選択有_TB
      OUT     M180  ; 送り 芯金干渉ﾌﾗｸﾞ
      MRD
      AND     X108A  ; LS73 ﾜｲﾊﾟｰ有
      OUT     M181  ; 送り ﾜｲﾊﾟｰ干渉ﾌﾗｸﾞ
      MRD
      LDI     X1064  ; LS9 ﾌﾟﾚｯｼｬｰ 開
      OR      X106B  ; LS4 ﾌﾟﾚｯｼｬｰﾀﾞｲ 後退(原点)
      OR      M7049  ; D70=201　干渉確認用接点
      OR      B12A  ; ﾘﾄﾗｸﾄﾌﾟﾚｯｼｬ連結中
      ANB
      OUT     M182  ; 送り ｽﾗｲﾄﾞﾌﾟﾚｯｼｬｰ干渉確認
      MPP
      AND     M180  ; 送り 芯金干渉ﾌﾗｸﾞ
      MPS
      ANDD<   D120 R20138  ; 送り前進可能位置 / 送り芯金干渉位置
      DMOV    R20138 D120
      MPP
      ANDD<=  D100 R20138  ; 送り現在値 / 送り芯金干渉位置
      ANDD=   D120 R20138  ; 送り前進可能位置 / 送り芯金干渉位置
      OUT     M175  ; 送り芯金干渉位置
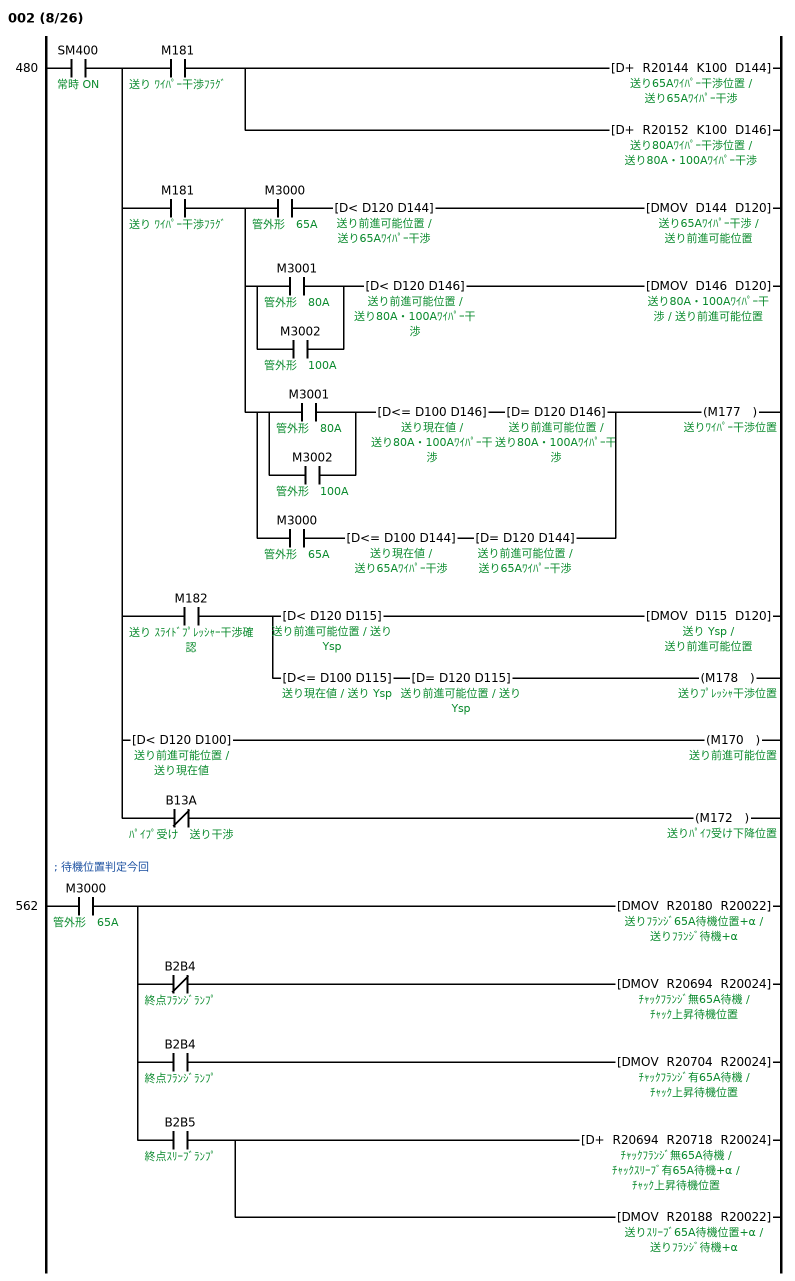
480   LD      SM400  ; 常時 ON
      MPS
      AND     M181  ; 送り ﾜｲﾊﾟｰ干渉ﾌﾗｸﾞ
      D+      R20144 K100 D144  ; 送り65Aﾜｲﾊﾟｰ干渉
      D+      R20152 K100 D146  ; 送り80A・100Aﾜｲﾊﾟｰ干渉
      MRD
      AND     M181  ; 送り ﾜｲﾊﾟｰ干渉ﾌﾗｸﾞ
      MPS
      AND     M3000  ; 管外形　65A
      ANDD<   D120 D144  ; 送り前進可能位置 / 送り65Aﾜｲﾊﾟｰ干渉
      DMOV    D144 D120
      MRD
      LD      M3001  ; 管外形　80A
      OR      M3002  ; 管外形　100A
      ANB
      ANDD<   D120 D146  ; 送り前進可能位置 / 送り80A・100Aﾜｲﾊﾟｰ干渉
      DMOV    D146 D120
      MPP
      LD      M3001  ; 管外形　80A
      OR      M3002  ; 管外形　100A
      ANDD<=  D100 D146  ; 送り現在値 / 送り80A・100Aﾜｲﾊﾟｰ干渉
      ANDD=   D120 D146  ; 送り前進可能位置 / 送り80A・100Aﾜｲﾊﾟｰ干渉
      LD      M3000  ; 管外形　65A
      ANDD<=  D100 D144  ; 送り現在値 / 送り65Aﾜｲﾊﾟｰ干渉
      ANDD=   D120 D144  ; 送り前進可能位置 / 送り65Aﾜｲﾊﾟｰ干渉
      ORB
      ANB
      OUT     M177  ; 送りﾜｲﾊﾟｰ干渉位置
      MRD
      AND     M182  ; 送り ｽﾗｲﾄﾞﾌﾟﾚｯｼｬｰ干渉確認
      MPS
      ANDD<   D120 D115  ; 送り前進可能位置 / 送り Ysp
      DMOV    D115 D120
      MPP
      ANDD<=  D100 D115  ; 送り現在値 / 送り Ysp
      ANDD=   D120 D115  ; 送り前進可能位置 / 送り Ysp
      OUT     M178  ; 送りﾌﾟﾚｯｼｬ干渉位置
      MRD
      ANDD<   D120 D100  ; 送り前進可能位置 / 送り現在値
      OUT     M170  ; 送り前進可能位置
      MPP
      ANI     B13A  ; ﾊﾟｲﾌﾟ受け　送り干渉
      OUT     M172  ; 送りﾊﾟｲﾌ受け下降位置
; 待機位置判定今回
562   LD      M3000  ; 管外形　65A
      DMOV    R20180 R20022  ; 送りﾌﾗﾝｼﾞ65A待機位置+α
      MPS
      ANI     B2B4  ; 終点ﾌﾗﾝｼﾞﾗﾝﾌﾟ
      DMOV    R20694 R20024  ; ﾁｬｯｸﾌﾗﾝｼﾞ無65A待機 / ﾁｬｯｸ上昇待機位置
      MRD
      AND     B2B4  ; 終点ﾌﾗﾝｼﾞﾗﾝﾌﾟ
      DMOV    R20704 R20024  ; ﾁｬｯｸﾌﾗﾝｼﾞ有65A待機
      MPP
      AND     B2B5  ; 終点ｽﾘｰﾌﾞﾗﾝﾌﾟ
      D+      R20694 R20718 R20024  ; ﾁｬｯｸｽﾘｰﾌﾞ有65A待機+α
      DMOV    R20188 R20022  ; 送りｽﾘｰﾌﾞ65A待機位置+α
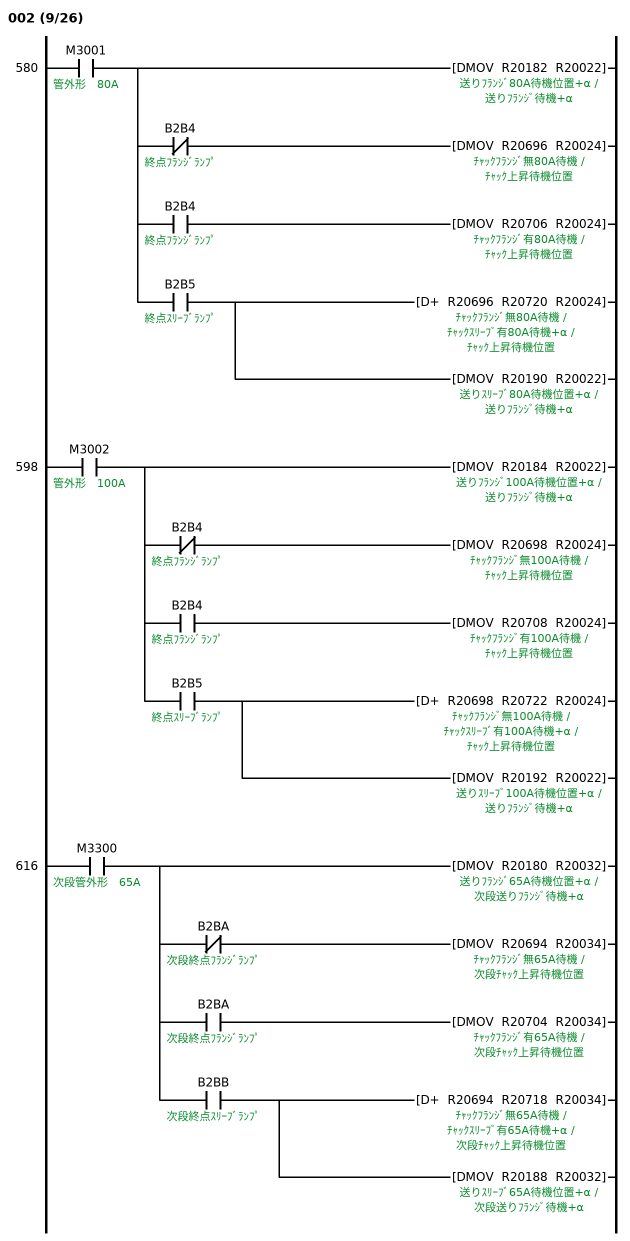
580   LD      M3001  ; 管外形　80A
      DMOV    R20182 R20022  ; 送りﾌﾗﾝｼﾞ80A待機位置+α
      MPS
      ANI     B2B4  ; 終点ﾌﾗﾝｼﾞﾗﾝﾌﾟ
      DMOV    R20696 R20024  ; ﾁｬｯｸﾌﾗﾝｼﾞ無80A待機
      MRD
      AND     B2B4  ; 終点ﾌﾗﾝｼﾞﾗﾝﾌﾟ
      DMOV    R20706 R20024  ; ﾁｬｯｸﾌﾗﾝｼﾞ有80A待機
      MPP
      AND     B2B5  ; 終点ｽﾘｰﾌﾞﾗﾝﾌﾟ
      D+      R20696 R20720 R20024  ; ﾁｬｯｸｽﾘｰﾌﾞ有80A待機+α
      DMOV    R20190 R20022  ; 送りｽﾘｰﾌﾞ80A待機位置+α
598   LD      M3002  ; 管外形　100A
      DMOV    R20184 R20022  ; 送りﾌﾗﾝｼﾞ100A待機位置+α
      MPS
      ANI     B2B4  ; 終点ﾌﾗﾝｼﾞﾗﾝﾌﾟ
      DMOV    R20698 R20024  ; ﾁｬｯｸﾌﾗﾝｼﾞ無100A待機
      MRD
      AND     B2B4  ; 終点ﾌﾗﾝｼﾞﾗﾝﾌﾟ
      DMOV    R20708 R20024  ; ﾁｬｯｸﾌﾗﾝｼﾞ有100A待機
      MPP
      AND     B2B5  ; 終点ｽﾘｰﾌﾞﾗﾝﾌﾟ
      D+      R20698 R20722 R20024  ; ﾁｬｯｸｽﾘｰﾌﾞ有100A待機+α
      DMOV    R20192 R20022  ; 送りｽﾘｰﾌﾞ100A待機位置+α
616   LD      M3300  ; 次段管外形　65A
      DMOV    R20180 R20032  ; 次段送りﾌﾗﾝｼﾞ待機+α
      MPS
      ANI     B2BA  ; 次段終点ﾌﾗﾝｼﾞﾗﾝﾌﾟ
      DMOV    R20694 R20034  ; 次段ﾁｬｯｸ上昇待機位置
      MRD
      AND     B2BA  ; 次段終点ﾌﾗﾝｼﾞﾗﾝﾌﾟ
      DMOV    R20704 R20034
      MPP
      AND     B2BB  ; 次段終点ｽﾘｰﾌﾞﾗﾝﾌﾟ
      D+      R20694 R20718 R20034
      DMOV    R20188 R20032
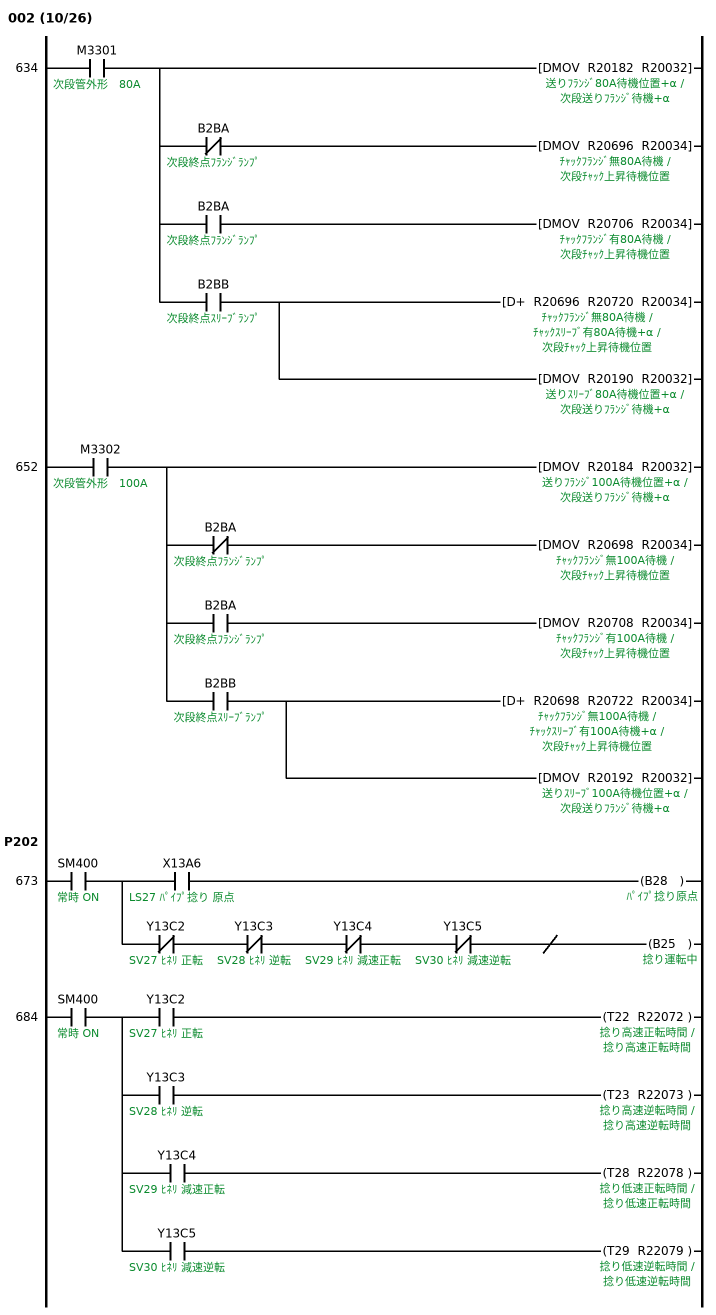
634   LD      M3301  ; 次段管外形　80A
      DMOV    R20182 R20032
      MPS
      ANI     B2BA  ; 次段終点ﾌﾗﾝｼﾞﾗﾝﾌﾟ
      DMOV    R20696 R20034
      MRD
      AND     B2BA  ; 次段終点ﾌﾗﾝｼﾞﾗﾝﾌﾟ
      DMOV    R20706 R20034
      MPP
      AND     B2BB  ; 次段終点ｽﾘｰﾌﾞﾗﾝﾌﾟ
      D+      R20696 R20720 R20034
      DMOV    R20190 R20032
652   LD      M3302  ; 次段管外形　100A
      DMOV    R20184 R20032
      MPS
      ANI     B2BA  ; 次段終点ﾌﾗﾝｼﾞﾗﾝﾌﾟ
      DMOV    R20698 R20034
      MRD
      AND     B2BA  ; 次段終点ﾌﾗﾝｼﾞﾗﾝﾌﾟ
      DMOV    R20708 R20034
      MPP
      AND     B2BB  ; 次段終点ｽﾘｰﾌﾞﾗﾝﾌﾟ
      D+      R20698 R20722 R20034
      DMOV    R20192 R20032
; 
      P202
673   LD      SM400  ; 常時 ON
      MPS
      AND     X13A6  ; LS27 ﾊﾟｲﾌﾟ捻り 原点
      OUT     B28  ; ﾊﾟｲﾌﾟ捻り原点
      MPP
      ANI     Y13C2  ; SV27 ﾋﾈﾘ 正転
      ANI     Y13C3  ; SV28 ﾋﾈﾘ 逆転
      ANI     Y13C4  ; SV29 ﾋﾈﾘ 減速正転
      ANI     Y13C5  ; SV30 ﾋﾈﾘ 減速逆転
      INV
      OUT     B25  ; 捻り運転中
684   LD      SM400  ; 常時 ON
      MPS
      AND     Y13C2  ; SV27 ﾋﾈﾘ 正転
      OUT     T22 R22072  ; 捻り高速正転時間 / 捻り高速正転時間
      MRD
      AND     Y13C3  ; SV28 ﾋﾈﾘ 逆転
      OUT     T23 R22073  ; 捻り高速逆転時間 / 捻り高速逆転時間
      MRD
      AND     Y13C4  ; SV29 ﾋﾈﾘ 減速正転
      OUT     T28 R22078  ; 捻り低速正転時間 / 捻り低速正転時間
      MPP
      AND     Y13C5  ; SV30 ﾋﾈﾘ 減速逆転
      OUT     T29 R22079  ; 捻り低速逆転時間 / 捻り低速逆転時間
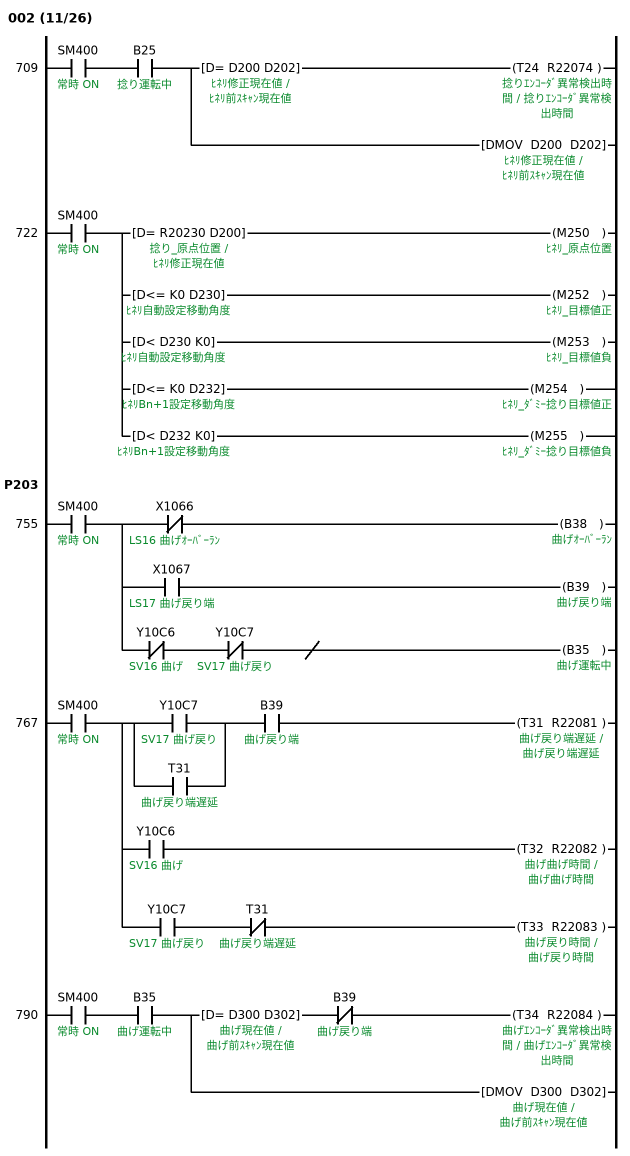
709   LD      SM400  ; 常時 ON
      AND     B25  ; 捻り運転中
      MPS
      ANDD=   D200 D202  ; ﾋﾈﾘ修正現在値 / ﾋﾈﾘ前ｽｷｬﾝ現在値
      OUT     T24 R22074  ; 捻りｴﾝｺｰﾀﾞ異常検出時間 / 捻りｴﾝｺｰﾀﾞ異常検出時間
      MPP
      DMOV    D200 D202
722   LD      SM400  ; 常時 ON
      MPS
      ANDD=   R20230 D200  ; 捻り_原点位置 / ﾋﾈﾘ修正現在値
      OUT     M250  ; ﾋﾈﾘ_原点位置
      MRD
      ANDD<=  K0 D230  ; ﾋﾈﾘ自動設定移動角度
      OUT     M252  ; ﾋﾈﾘ_目標値正
      MRD
      ANDD<   D230 K0  ; ﾋﾈﾘ自動設定移動角度
      OUT     M253  ; ﾋﾈﾘ_目標値負
      MRD
      ANDD<=  K0 D232  ; ﾋﾈﾘBn+1設定移動角度
      OUT     M254  ; ﾋﾈﾘ_ﾀﾞﾐｰ捻り目標値正
      MPP
      ANDD<   D232 K0  ; ﾋﾈﾘBn+1設定移動角度
      OUT     M255  ; ﾋﾈﾘ_ﾀﾞﾐｰ捻り目標値負
; 
      P203
755   LD      SM400  ; 常時 ON
      MPS
      ANI     X1066  ; LS16 曲げｵｰﾊﾞｰﾗﾝ
      OUT     B38  ; 曲げｵｰﾊﾞｰﾗﾝ
      MRD
      AND     X1067  ; LS17 曲げ戻り端
      OUT     B39  ; 曲げ戻り端
      MPP
      ANI     Y10C6  ; SV16 曲げ
      ANI     Y10C7  ; SV17 曲げ戻り
      INV
      OUT     B35  ; 曲げ運転中
767   LD      SM400  ; 常時 ON
      MPS
      LD      Y10C7  ; SV17 曲げ戻り
      OR      T31  ; 曲げ戻り端遅延
      ANB
      AND     B39  ; 曲げ戻り端
      OUT     T31 R22081  ; 曲げ戻り端遅延 / 曲げ戻り端遅延
      MRD
      AND     Y10C6  ; SV16 曲げ
      OUT     T32 R22082  ; 曲げ曲げ時間 / 曲げ曲げ時間
      MPP
      AND     Y10C7  ; SV17 曲げ戻り
      ANI     T31  ; 曲げ戻り端遅延
      OUT     T33 R22083  ; 曲げ戻り時間 / 曲げ戻り時間
790   LD      SM400  ; 常時 ON
      AND     B35  ; 曲げ運転中
      MPS
      ANDD=   D300 D302  ; 曲げ現在値 / 曲げ前ｽｷｬﾝ現在値
      ANI     B39  ; 曲げ戻り端
      OUT     T34 R22084  ; 曲げｴﾝｺｰﾀﾞ異常検出時間 / 曲げｴﾝｺｰﾀﾞ異常検出時間
      MPP
      DMOV    D300 D302
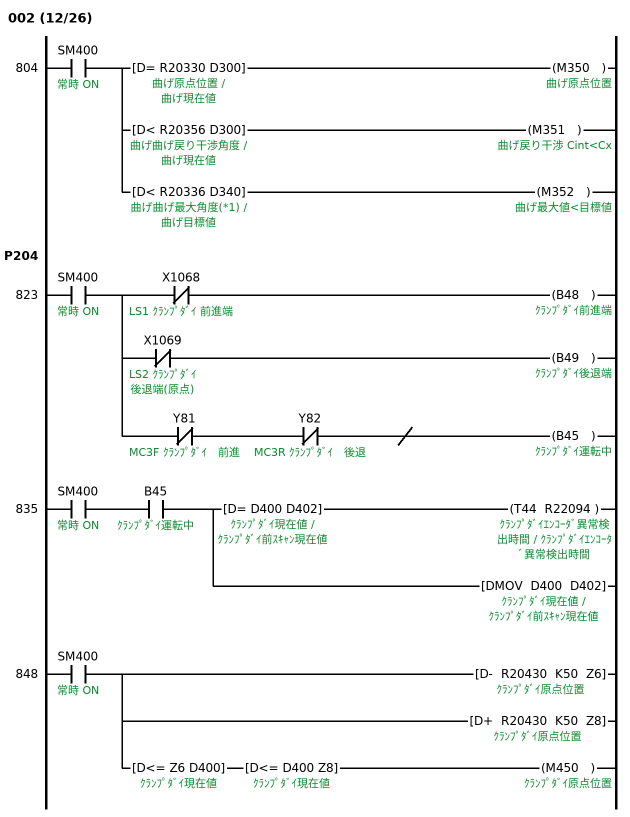
804   LD      SM400  ; 常時 ON
      MPS
      ANDD=   R20330 D300  ; 曲げ原点位置 / 曲げ現在値
      OUT     M350  ; 曲げ原点位置
      MRD
      ANDD<   R20356 D300  ; 曲げ曲げ戻り干渉角度 / 曲げ現在値
      OUT     M351  ; 曲げ戻り干渉 Cint<Cx
      MPP
      ANDD<   R20336 D340  ; 曲げ曲げ最大角度(*1) / 曲げ目標値
      OUT     M352  ; 曲げ最大値<目標値
; 
      P204
823   LD      SM400  ; 常時 ON
      MPS
      ANI     X1068  ; LS1 ｸﾗﾝﾌﾟﾀﾞｲ 前進端
      OUT     B48  ; ｸﾗﾝﾌﾟﾀﾞｲ前進端
      MRD
      ANI     X1069  ; LS2 ｸﾗﾝﾌﾟﾀﾞｲ 後退端(原点)
      OUT     B49  ; ｸﾗﾝﾌﾟﾀﾞｲ後退端
      MPP
      ANI     Y81  ; MC3F ｸﾗﾝﾌﾟﾀﾞｲ　前進
      ANI     Y82  ; MC3R ｸﾗﾝﾌﾟﾀﾞｲ　後退
      INV
      OUT     B45  ; ｸﾗﾝﾌﾟﾀﾞｲ運転中
835   LD      SM400  ; 常時 ON
      AND     B45  ; ｸﾗﾝﾌﾟﾀﾞｲ運転中
      MPS
      ANDD=   D400 D402  ; ｸﾗﾝﾌﾟﾀﾞｲ現在値 / ｸﾗﾝﾌﾟﾀﾞｲ前ｽｷｬﾝ現在値
      OUT     T44 R22094  ; ｸﾗﾝﾌﾟﾀﾞｲｴﾝｺｰﾀﾞ異常検出時間 / ｸﾗﾝﾌﾟﾀﾞｲｴﾝｺｰﾀﾞ異常検出時間
      MPP
      DMOV    D400 D402
848   LD      SM400  ; 常時 ON
      D-      R20430 K50 Z6  ; ｸﾗﾝﾌﾟﾀﾞｲ原点位置
      D+      R20430 K50 Z8
      ANDD<=  Z6 D400  ; ｸﾗﾝﾌﾟﾀﾞｲ現在値
      ANDD<=  D400 Z8  ; ｸﾗﾝﾌﾟﾀﾞｲ現在値
      OUT     M450  ; ｸﾗﾝﾌﾟﾀﾞｲ原点位置
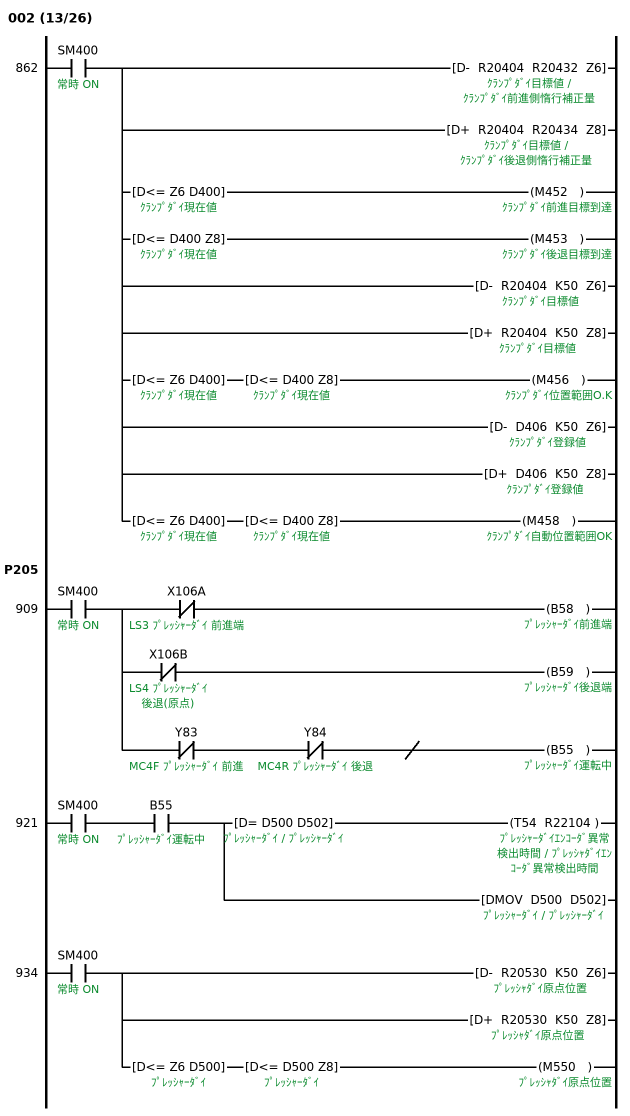
862   LD      SM400  ; 常時 ON
      D-      R20404 R20432 Z6  ; ｸﾗﾝﾌﾟﾀﾞｲ目標値 / ｸﾗﾝﾌﾟﾀﾞｲ前進側惰行補正量
      D+      R20404 R20434 Z8  ; ｸﾗﾝﾌﾟﾀﾞｲ後退側惰行補正量
      MPS
      ANDD<=  Z6 D400  ; ｸﾗﾝﾌﾟﾀﾞｲ現在値
      OUT     M452  ; ｸﾗﾝﾌﾟﾀﾞｲ前進目標到達
      MRD
      ANDD<=  D400 Z8  ; ｸﾗﾝﾌﾟﾀﾞｲ現在値
      OUT     M453  ; ｸﾗﾝﾌﾟﾀﾞｲ後退目標到達
      MPP
      D-      R20404 K50 Z6
      D+      R20404 K50 Z8
      MPS
      ANDD<=  Z6 D400  ; ｸﾗﾝﾌﾟﾀﾞｲ現在値
      ANDD<=  D400 Z8  ; ｸﾗﾝﾌﾟﾀﾞｲ現在値
      OUT     M456  ; ｸﾗﾝﾌﾟﾀﾞｲ位置範囲O.K
      MPP
      D-      D406 K50 Z6  ; ｸﾗﾝﾌﾟﾀﾞｲ登録値
      D+      D406 K50 Z8
      ANDD<=  Z6 D400  ; ｸﾗﾝﾌﾟﾀﾞｲ現在値
      ANDD<=  D400 Z8  ; ｸﾗﾝﾌﾟﾀﾞｲ現在値
      OUT     M458  ; ｸﾗﾝﾌﾟﾀﾞｲ自動位置範囲OK
; 
      P205
909   LD      SM400  ; 常時 ON
      MPS
      ANI     X106A  ; LS3 ﾌﾟﾚｯｼｬｰﾀﾞｲ 前進端
      OUT     B58  ; ﾌﾟﾚｯｼｬｰﾀﾞｲ前進端
      MRD
      ANI     X106B  ; LS4 ﾌﾟﾚｯｼｬｰﾀﾞｲ 後退(原点)
      OUT     B59  ; ﾌﾟﾚｯｼｬｰﾀﾞｲ後退端
      MPP
      ANI     Y83  ; MC4F ﾌﾟﾚｯｼｬｰﾀﾞｲ 前進
      ANI     Y84  ; MC4R ﾌﾟﾚｯｼｬｰﾀﾞｲ 後退
      INV
      OUT     B55  ; ﾌﾟﾚｯｼｬｰﾀﾞｲ運転中
921   LD      SM400  ; 常時 ON
      AND     B55  ; ﾌﾟﾚｯｼｬｰﾀﾞｲ運転中
      MPS
      ANDD=   D500 D502  ; ﾌﾟﾚｯｼｬｰﾀﾞｲ / ﾌﾟﾚｯｼｬｰﾀﾞｲ
      OUT     T54 R22104  ; ﾌﾟﾚｯｼｬｰﾀﾞｲｴﾝｺｰﾀﾞ異常検出時間 / ﾌﾟﾚｯｼｬﾀﾞｲｴﾝｺｰﾀﾞ異常検出時間
      MPP
      DMOV    D500 D502
934   LD      SM400  ; 常時 ON
      D-      R20530 K50 Z6  ; ﾌﾟﾚｯｼｬﾀﾞｲ原点位置
      D+      R20530 K50 Z8
      ANDD<=  Z6 D500  ; ﾌﾟﾚｯｼｬｰﾀﾞｲ
      ANDD<=  D500 Z8  ; ﾌﾟﾚｯｼｬｰﾀﾞｲ
      OUT     M550  ; ﾌﾟﾚｯｼｬﾀﾞｲ原点位置
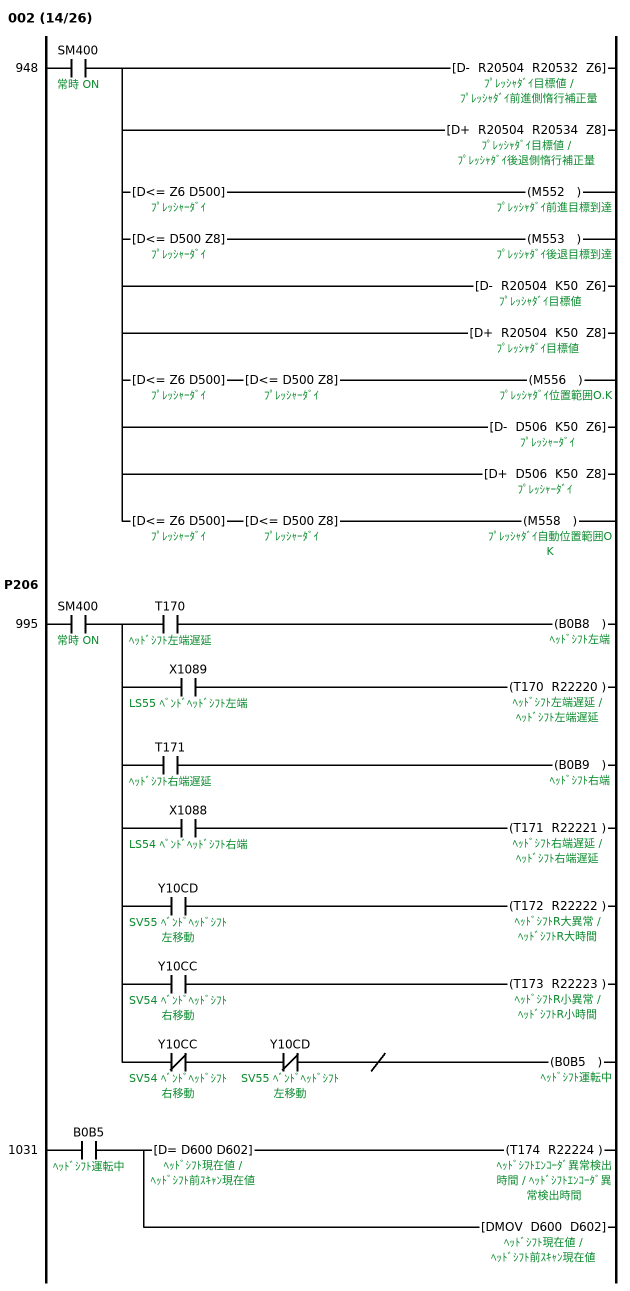
948   LD      SM400  ; 常時 ON
      D-      R20504 R20532 Z6  ; ﾌﾟﾚｯｼｬﾀﾞｲ目標値 / ﾌﾟﾚｯｼｬﾀﾞｲ前進側惰行補正量
      D+      R20504 R20534 Z8  ; ﾌﾟﾚｯｼｬﾀﾞｲ後退側惰行補正量
      MPS
      ANDD<=  Z6 D500  ; ﾌﾟﾚｯｼｬｰﾀﾞｲ
      OUT     M552  ; ﾌﾟﾚｯｼｬﾀﾞｲ前進目標到達
      MRD
      ANDD<=  D500 Z8  ; ﾌﾟﾚｯｼｬｰﾀﾞｲ
      OUT     M553  ; ﾌﾟﾚｯｼｬﾀﾞｲ後退目標到達
      MPP
      D-      R20504 K50 Z6
      D+      R20504 K50 Z8
      MPS
      ANDD<=  Z6 D500  ; ﾌﾟﾚｯｼｬｰﾀﾞｲ
      ANDD<=  D500 Z8  ; ﾌﾟﾚｯｼｬｰﾀﾞｲ
      OUT     M556  ; ﾌﾟﾚｯｼｬﾀﾞｲ位置範囲O.K
      MPP
      D-      D506 K50 Z6  ; ﾌﾟﾚｯｼｬｰﾀﾞｲ
      D+      D506 K50 Z8
      ANDD<=  Z6 D500  ; ﾌﾟﾚｯｼｬｰﾀﾞｲ
      ANDD<=  D500 Z8  ; ﾌﾟﾚｯｼｬｰﾀﾞｲ
      OUT     M558  ; ﾌﾟﾚｯｼｬﾀﾞｲ自動位置範囲OK
; 
      P206
995   LD      SM400  ; 常時 ON
      MPS
      AND     T170  ; ﾍｯﾄﾞｼﾌﾄ左端遅延
      OUT     B0B8  ; ﾍｯﾄﾞｼﾌﾄ左端
      MRD
      AND     X1089  ; LS55 ﾍﾞﾝﾄﾞﾍｯﾄﾞｼﾌﾄ左端
      OUT     T170 R22220  ; ﾍｯﾄﾞｼﾌﾄ左端遅延 / ﾍｯﾄﾞｼﾌﾄ左端遅延
      MRD
      AND     T171  ; ﾍｯﾄﾞｼﾌﾄ右端遅延
      OUT     B0B9  ; ﾍｯﾄﾞｼﾌﾄ右端
      MRD
      AND     X1088  ; LS54 ﾍﾞﾝﾄﾞﾍｯﾄﾞｼﾌﾄ右端
      OUT     T171 R22221  ; ﾍｯﾄﾞｼﾌﾄ右端遅延 / ﾍｯﾄﾞｼﾌﾄ右端遅延
      MRD
      AND     Y10CD  ; SV55 ﾍﾞﾝﾄﾞﾍｯﾄﾞｼﾌﾄ 左移動
      OUT     T172 R22222  ; ﾍｯﾄﾞｼﾌﾄR大異常 / ﾍｯﾄﾞｼﾌﾄR大時間
      MRD
      AND     Y10CC  ; SV54 ﾍﾞﾝﾄﾞﾍｯﾄﾞｼﾌﾄ 右移動
      OUT     T173 R22223  ; ﾍｯﾄﾞｼﾌﾄR小異常 / ﾍｯﾄﾞｼﾌﾄR小時間
      MPP
      ANI     Y10CC  ; SV54 ﾍﾞﾝﾄﾞﾍｯﾄﾞｼﾌﾄ 右移動
      ANI     Y10CD  ; SV55 ﾍﾞﾝﾄﾞﾍｯﾄﾞｼﾌﾄ 左移動
      INV
      OUT     B0B5  ; ﾍｯﾄﾞｼﾌﾄ運転中
1031  LD      B0B5  ; ﾍｯﾄﾞｼﾌﾄ運転中
      MPS
      ANDD=   D600 D602  ; ﾍｯﾄﾞｼﾌﾄ現在値 / ﾍｯﾄﾞｼﾌﾄ前ｽｷｬﾝ現在値
      OUT     T174 R22224  ; ﾍｯﾄﾞｼﾌﾄｴﾝｺｰﾀﾞ異常検出時間 / ﾍｯﾄﾞｼﾌﾄｴﾝｺｰﾀﾞ異常検出時間
      MPP
      DMOV    D600 D602
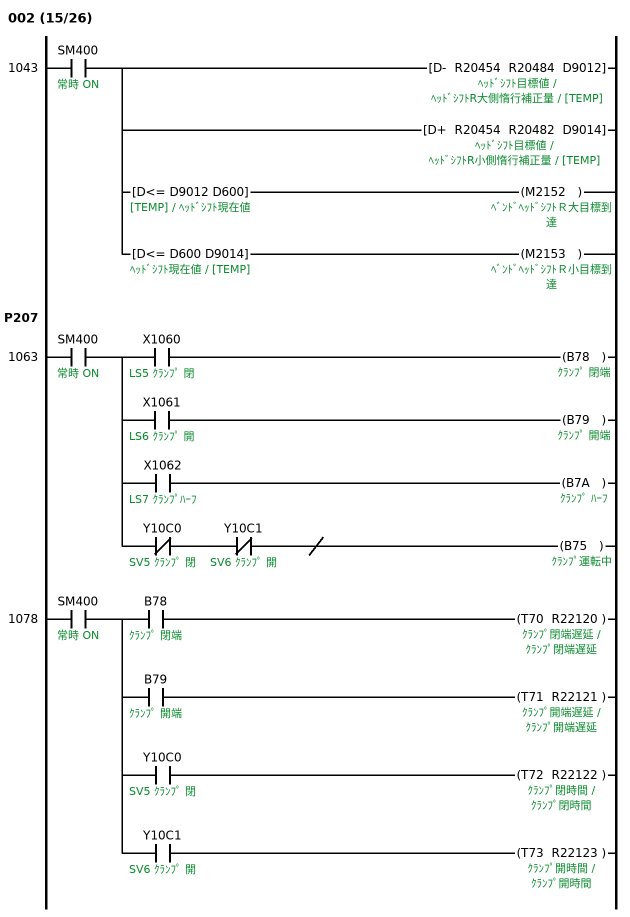
1043  LD      SM400  ; 常時 ON
      D-      R20454 R20484 D9012  ; ﾍｯﾄﾞｼﾌﾄ目標値 / ﾍｯﾄﾞｼﾌﾄR大側惰行補正量 / [TEMP]
      D+      R20454 R20482 D9014  ; ﾍｯﾄﾞｼﾌﾄR小側惰行補正量 / [TEMP]
      MPS
      ANDD<=  D9012 D600  ; [TEMP] / ﾍｯﾄﾞｼﾌﾄ現在値
      OUT     M2152  ; ﾍﾞﾝﾄﾞﾍｯﾄﾞｼﾌﾄＲ大目標到達
      MPP
      ANDD<=  D600 D9014  ; ﾍｯﾄﾞｼﾌﾄ現在値 / [TEMP]
      OUT     M2153  ; ﾍﾞﾝﾄﾞﾍｯﾄﾞｼﾌﾄＲ小目標到達
; 
      P207
1063  LD      SM400  ; 常時 ON
      MPS
      AND     X1060  ; LS5 ｸﾗﾝﾌﾟ 閉
      OUT     B78  ; ｸﾗﾝﾌﾟ 閉端
      MRD
      AND     X1061  ; LS6 ｸﾗﾝﾌﾟ 開
      OUT     B79  ; ｸﾗﾝﾌﾟ 開端
      MRD
      AND     X1062  ; LS7 ｸﾗﾝﾌﾟﾊｰﾌ
      OUT     B7A  ; ｸﾗﾝﾌﾟ ﾊｰﾌ
      MPP
      ANI     Y10C0  ; SV5 ｸﾗﾝﾌﾟ 閉
      ANI     Y10C1  ; SV6 ｸﾗﾝﾌﾟ 開
      INV
      OUT     B75  ; ｸﾗﾝﾌﾟ運転中
1078  LD      SM400  ; 常時 ON
      MPS
      AND     B78  ; ｸﾗﾝﾌﾟ 閉端
      OUT     T70 R22120  ; ｸﾗﾝﾌﾟ閉端遅延 / ｸﾗﾝﾌﾟ閉端遅延
      MRD
      AND     B79  ; ｸﾗﾝﾌﾟ 開端
      OUT     T71 R22121  ; ｸﾗﾝﾌﾟ開端遅延 / ｸﾗﾝﾌﾟ開端遅延
      MRD
      AND     Y10C0  ; SV5 ｸﾗﾝﾌﾟ 閉
      OUT     T72 R22122  ; ｸﾗﾝﾌﾟ閉時間 / ｸﾗﾝﾌﾟ閉時間
      MPP
      AND     Y10C1  ; SV6 ｸﾗﾝﾌﾟ 開
      OUT     T73 R22123  ; ｸﾗﾝﾌﾟ開時間 / ｸﾗﾝﾌﾟ開時間
; 
      P208
